TYPE "UDT_ModuleState"
TITLE = UDT_ModuleState
VERSION : 0.1
//User-defined structure of module states.
   STRUCT
      Configured { ExternalAccessible := 'False'; ExternalVisible := 'False'; ExternalWritable := 'False'} : Bool;   // Module configured
      Exist { ExternalAccessible := 'False'; ExternalVisible := 'False'; ExternalWritable := 'False'} : Bool;   // Module exist
      Error { ExternalAccessible := 'False'; ExternalVisible := 'False'; ExternalWritable := 'False'} : Bool;   // Module has error
   END_STRUCT;

END_TYPE

TYPE "UDT_DeviceState"
TITLE = UDT_DeviceState
VERSION : 0.1
//User-defined structure of device states.
   STRUCT
      Configure { ExternalAccessible := 'False'; ExternalVisible := 'False'; ExternalWritable := 'False'} : Bool;   // Device configured in TIA Portal hardware
      Exist { ExternalAccessible := 'False'; ExternalVisible := 'False'; ExternalWritable := 'False'} : Bool;   // Device physically connected
      Error { ExternalAccessible := 'False'; ExternalVisible := 'False'; ExternalWritable := 'False'} : Bool;   // Device has an error
      ProfinetNumber : UInt;   // Profinet slave number
      HW_ID : UInt;   // Device's HW_ID
      PNDeviceName : String;   // Device's project name
   END_STRUCT;

END_TYPE

TYPE "UDT_GINDHL"
VERSION : 0.1
   STRUCT
      ObjectID : String[10];   // Object ID
      VID : String[16];   // Virtual Item Identifier (VID)
      PieceID : String[40];   // Piece ID barcodes
      SortStrategy : String[1];   // Sort Strategy 1 - Highest priority available , 2 - Nearest
      ParcelReject { ExternalAccessible := 'False'; ExternalVisible := 'False'; ExternalWritable := 'False'} : Bool;   // True - Parcel reject
      Destination : Array[1..6] of Struct   // Destination
         ID : UInt;   // ID
         SortCommandActive { ExternalAccessible := 'False'; ExternalVisible := 'False'; ExternalWritable := 'False'} : Bool;   // Sort command
         ParcelSorted { ExternalAccessible := 'False'; ExternalVisible := 'False'; ExternalWritable := 'False'} : Bool;   // Parcel sorted
         Rejected { ExternalAccessible := 'False'; ExternalVisible := 'False'; ExternalWritable := 'False'} : Bool;   // Parcel rejected
         Reason : Int;   // Reason
      END_STRUCT;
      ParcelLocation : Struct   // Parcel Location
         Current : UInt;   // Current
         Last : UInt;   // Last
         Sort : UInt;   // Sort
      END_STRUCT;
      MFCMessage : Struct   // MFC Sort messages
         Sent : Struct   // Messages sent from the PLC to the MFC system
            SortResult { ExternalAccessible := 'False'; ExternalVisible := 'False'; ExternalWritable := 'False'} : Bool;   // Message Sort Result
            VIDResponse { ExternalAccessible := 'False'; ExternalVisible := 'False'; ExternalWritable := 'False'} : Bool;   // Message VID Response
            ScanReset { ExternalAccessible := 'False'; ExternalVisible := 'False'; ExternalWritable := 'False'} : Bool;   // Message Scan Reset
            XrayResult { ExternalAccessible := 'False'; ExternalVisible := 'False'; ExternalWritable := 'False'} : Bool;   // Message Xray result
            ParcelRegInfo { ExternalAccessible := 'False'; ExternalVisible := 'False'; ExternalWritable := 'False'} : Bool;   // Message Xray registration info
         END_STRUCT;
         Received : Struct   // Messages received from the MFC system to the PLC
            RejectParcel { ExternalAccessible := 'False'; ExternalVisible := 'False'; ExternalWritable := 'False'} : Bool;   // Message Reject Parcel
            Destination { ExternalAccessible := 'False'; ExternalVisible := 'False'; ExternalWritable := 'False'} : Bool;   // Message Destination
            DestinationResent { ExternalAccessible := 'False'; ExternalVisible := 'False'; ExternalWritable := 'False'} : Bool;   // Message Destination Resent
            TemporaryParcelIdentifier { ExternalAccessible := 'False'; ExternalVisible := 'False'; ExternalWritable := 'False'} : Bool;   // Message Temporary Parcel Identifier
            XrayRegistrationInfo { ExternalAccessible := 'False'; ExternalVisible := 'False'; ExternalWritable := 'False'} : Bool;
         END_STRUCT;
      END_STRUCT;
      Xray : Struct   // Xray data structure
         RoutingCode : String[2];   // Routing code
         Group : String[1];   // The group field is used to identify the group of the operator decisions came from in a
         Level : String[1];   // Level field is used to identify which level the operator decision came from in a
         Result : String[1];   // Results can be indicated with the following:A = Accept, R = Reject, U = Unavailable (Timeout), Z = High Threat
         BagIDMessage : Struct   // Message from PLC to Xray
            MessagePrepared { ExternalAccessible := 'False'; ExternalVisible := 'False'; ExternalWritable := 'False'} : Bool;   // The message is prepared and ready to send
            WrongMessageStructure { ExternalAccessible := 'False'; ExternalVisible := 'False'; ExternalWritable := 'False'} : Bool;   // The message has wrong structure
            Sent { ExternalAccessible := 'False'; ExternalVisible := 'False'; ExternalWritable := 'False'} : Bool;   // The message sent by PLC to Xray
            SentTime : String;   // Time when message sent by PLC to Xray
            NotSent { ExternalAccessible := 'False'; ExternalVisible := 'False'; ExternalWritable := 'False'} : Bool;   // The message was not sent from the PLC
            Received { ExternalAccessible := 'False'; ExternalVisible := 'False'; ExternalWritable := 'False'} : Bool;   // The message received by Xray
            TimeReceived : String;   // Time when message received by Xray
            NotReceived { ExternalAccessible := 'False'; ExternalVisible := 'False'; ExternalWritable := 'False'} : Bool;   // The message did not reach Xray
         END_STRUCT;
         DecisionMessage : Struct   // Message from Xray to PLC
            Received { ExternalAccessible := 'False'; ExternalVisible := 'False'; ExternalWritable := 'False'} : Bool;   // The message received by PLC
            ReceivedTime : String;   // The message received by PLC
            NotReceivedOnTime { ExternalAccessible := 'False'; ExternalVisible := 'False'; ExternalWritable := 'False'} : Bool;   // The message did not reach PLC
         END_STRUCT;
      END_STRUCT;
   END_STRUCT;

END_TYPE

TYPE "UDT_GINFedEx"
VERSION : 0.1
   STRUCT
      Timestamp : String[17];   // Local time timestamp
      TimeZoneDesignator : String[5];   // Time zone designator
      PackageEntrancePoint : String[14];   // Entrance point, where LLC starts tracking the parcel.
      PackageEntranceState : String[1];   // Entrance state
      PackageExitPoint : String[14];   // Exit point name, where LLC reports the last known tracking point.
      PackageExitState : String[1];   // Exit point state when LLC reports the last known tracking point.
      PalletType : String[2];   // Pallet code for different type of pallets on the market
      Mask : String[1];   // Flag to indicate that a pallet has been mask.
      CellNumber : String[4];   // Tray/Cell number (for loop sorters) or generated by LLC (on line sorters).
      CellsOccupied : String[1];   // Cells occupied by the piece for loop sorters.
      ImageID : String[6];   // Image ID number created by the ADC system.
      ScanUnitType : String[1];   // Scan unit type
      ADCSystemID : String[15];   // Number assigned by the ADC system
      PackageID : String[15];   // Number assigned by the LLC system
      LLCSystemID : String[15];
      HLCPackageID : String[10];   // Unique number for the specific package during it stays in HLC system.
      HLCResultCode : String[16];   // Result code based on processing of the scan event messages.
      ShipmentID : String[6];   // Consignment id of the parcel.
      WeightStatus : String[1];   // Status to indicate if the parcel/pallet has weight on the system.
      ActualDestination : String[6];   // Location code value that describes the actual disposition of the package.
      Destination1 : String[6];   // Location code value that describes where the package should go (Diverter Number).
      Destination2 : String[6];   // Location code value that describes where the package should go (Diverter Number).
      Destination3 : String[6];   // Location code value that describes where the package should go (Diverter Number).
      Destination4 : String[6];   // Location code value that describes where the package should go (Diverter Number).
      Destination5 : String[6];   // Location code value that describes where the package should go (Diverter Number).
      CutOffTimeDestination1 : String[5];   // Cut Off Time in Local Time.
      CutOffTimeDestination2 : String[5];   // Cut Off Time in Local Time.
      CutOffTimeDestination3 : String[5];   // Cut Off Time in Local Time.
      CutOffTimeDestination4 : String[5];   // Cut Off Time in Local Time.
      CutOffTimeDestination5 : String[5];   // Cut Off Time in Local Time.
      ReasonCode1 : String[8];   // Management Code value that describes the result of attempting to route the package to the Destination
      ReasonCode2 : String[8];   // Management Code value that describes the result of attempting to route the package to the Destination
      ReasonCode3 : String[8];   // Management Code value that describes the result of attempting to route the package to the Destination
      ReasonCode4 : String[8];   // Management Code value that describes the result of attempting to route the package to the Destination
      ReasonCode5 : String[8];   // Management Code value that describes the result of attempting to route the package to the Destination
      HLCDataText : String[20];   // Free text for future use.
      Customs : String[1];   // Need to be checked by customs
      DIMSystemID : String[15];   // Identifier of dimensioning system.
      DIMStatus : String[5];   // Basic diagnostic information from the dimensioning system at the moment of the measurement.
      PackageDimLength : String[6];   // Length dimension of package in resolution of dim system.
      PackageDimWidth : String[6];   // Width dimension of package in resolution of dim system.
      PackageDimHeight : String[6];   // Height dimension of package in resolution of dim system.
      DIMUOM : String[2];   // Unit of measure of the package dimensions.
      DimLFTstatusCode : String[8];   // Dimension LFT status code.
      DimConfidence : String[2];   // The level of assurance for the correct dimensions.
      DimensionSource : String[1];   // For combined camera/laser dim acquisition devices. It indicates type of capturing mode
      AlibiDims : String[25];   // Alibi for Dimensions
      SCLSystemID : String[15];   // Identifier of weight scale.
      SCLStatus : String[5];   // Basic diagnostic information from the weight scale system.
      SCLWT : String[6];   // Scale weight of package in resolution of scale system.
      SCLWTUOM : String[2];   // Unit of measurement for Weight
      SCLLFTStatusCode : String[2];   // Scale LFT status code.
      AlibiWeight : String[25];   // Alibi for Weight
      ReasonCode : String[1];   // This code should be used when the SI message has some defect.
      Stackable : String[1];   // If stackable recognition is enabled, Y or N
      Stickerstype : String[2];   // When optical recognition is used to sort
      FlyingDocument : String[1];   // Status to confirm if the document/flyer is prone to fly off the sorter.
      ModeofOperation : String[1];   // Camera Tunnel operational mode format:
      CameraHeadstatus : String[2];   // Diagnostic information on camera/laser heads performing barcode reads.
      PackageDataTruncated : String[1];   // Y = Full length of barcode data exceeds 9999 bytes, data truncated
      TotalBarcodeDataLength : String[4];   // Length of all barcode data that was sent in bytes;
      Barcode1Identification : String[3];   // Barcode identifier code.
      Barcode1status : String[2];   // Barcode confidence factor
      Barcode1datalength : String[4];   // String length of barcode data in bytes; inclusive of this field. Use 0054 as a fixed value
      Barcode1data : String[50];   // Highest priority barcode
      Barcode2Identification : String[3];   // Barcode identifier code.
      Barcode2status : String[2];   // Barcode confidence factor
      Barcode2datalength : String[4];   // String length of barcode data in bytes; inclusive of this field. Use 0054 as a fixed value
      Barcode2data : String[50];   // Highest priority barcode
      Barcode3Identification : String[3];   // Barcode identifier code.
      Barcode3status : String[2];   // Barcode confidence factor
      Barcode3datalength : String[4];   // String length of barcode data in bytes; inclusive of this field. Use 0054 as a fixed value
      Barcode3data : String[50];   // Highest priority barcode
      BarcodeIdentification : String[3];   // Barcode identifier code.
      Barcodestatus : String[2];   // Barcode confidence factor
      Barcodedatalength : String[4];   // String length of barcode data in bytes
      Barcodedata : String[50];   // Sortation barcode
      CustomerID : DInt;   // 6 digits SequentialID (NNNNNN)
      AreaNumber : String[2];   // Package Sequence ID "Area Number"
      PurgeEnabled { ExternalAccessible := 'False'; ExternalVisible := 'False'; ExternalWritable := 'False'} : Bool;   // Purge enabled for parcel: destination overwritten with Purge destination
   END_STRUCT;

END_TYPE

TYPE "UDT_GINStandard"
VERSION : 0.1
   STRUCT
      Destination : Array[0..20] of DInt;   // Destination
      Identification : Struct   // Barcode identification
         GoodRead { ExternalAccessible := 'False'; ExternalVisible := 'False'; ExternalWritable := 'False'} : Bool;   // Barcode read was succesful
         NoRead { ExternalAccessible := 'False'; ExternalVisible := 'False'; ExternalWritable := 'False'} : Bool;   // Barcode read was unsuccesful
         MultiRead { ExternalAccessible := 'False'; ExternalVisible := 'False'; ExternalWritable := 'False'} : Bool;   // Multiple Barcodes were detected
         Barcode : Array[0..10] of Char;   // Barcode values
      END_STRUCT;
      GinAssigned { ExternalAccessible := 'False'; ExternalVisible := 'False'; ExternalWritable := 'False'} : Bool;   // GIN is assigned to package
      Lost { ExternalAccessible := 'False'; ExternalVisible := 'False'; ExternalWritable := 'False'} : Bool;   // Lost in tracking
      Length : Int;   // Length in mm
      Width : Int;   // Width in mm
      Height : Int;   // Height in mm
      Weight : DInt;   // Weight in g
      PkgTooLong { ExternalAccessible := 'False'; ExternalVisible := 'False'; ExternalWritable := 'False'} : Bool;   // Package is too long
      PkgTooSmall { ExternalAccessible := 'False'; ExternalVisible := 'False'; ExternalWritable := 'False'} : Bool;   // Package is too small
      PkgTooHigh { ExternalAccessible := 'False'; ExternalVisible := 'False'; ExternalWritable := 'False'} : Bool;   // Package is too high
      PkgOverWeight { ExternalAccessible := 'False'; ExternalVisible := 'False'; ExternalWritable := 'False'} : Bool;   // Package is over weight
      TrailingGap : Int;   // Trailing gap size in cm between the package
      LeadingGap : Int;   // Leading gap size in cm between the package
      NrOfRecirculations : Int;   // Number of recirculations
      DestReqSend { ExternalAccessible := 'False'; ExternalVisible := 'False'; ExternalWritable := 'False'} : Bool;   // Destination request sent to high level
      DestRcv { ExternalAccessible := 'False'; ExternalVisible := 'False'; ExternalWritable := 'False'} : Bool;   // Destination received from high level
      SortStatus : Struct   // Sort status of the package
         DivertDestination : Int;   // Destination to which the package is diverted
         GoodDivert { ExternalAccessible := 'False'; ExternalVisible := 'False'; ExternalWritable := 'False'} : Bool;   // Package diverted
         FailedDivert { ExternalAccessible := 'False'; ExternalVisible := 'False'; ExternalWritable := 'False'} : Bool;   // Package failed to divert
         NoDivert : Bool := TRUE;   // Divert is not activated
         NoDivertCause : Struct   // Cause for no divert
            ChuteJam { ExternalAccessible := 'False'; ExternalVisible := 'False'; ExternalWritable := 'False'} : Bool;   // Chute is jammed
            ChuteFull { ExternalAccessible := 'False'; ExternalVisible := 'False'; ExternalWritable := 'False'} : Bool;   // Chute is full
            NoRTR { ExternalAccessible := 'False'; ExternalVisible := 'False'; ExternalWritable := 'False'} : Bool;   // Downstream conveyor is not ready to receive
            DestDisabled { ExternalAccessible := 'False'; ExternalVisible := 'False'; ExternalWritable := 'False'} : Bool;   // Destination is disabled
            TrayDisabled { ExternalAccessible := 'False'; ExternalVisible := 'False'; ExternalWritable := 'False'} : Bool;   // Tray is disabled
            SorterNotAtSpeed { ExternalAccessible := 'False'; ExternalVisible := 'False'; ExternalWritable := 'False'} : Bool;   // Sorter is not at speed
            LeadingGapError { ExternalAccessible := 'False'; ExternalVisible := 'False'; ExternalWritable := 'False'} : Bool;   // Gap size with downstream parcel is not enough
            TrailingGapError { ExternalAccessible := 'False'; ExternalVisible := 'False'; ExternalWritable := 'False'} : Bool;   // Gap size with upstream parcel is not enough
            PkgTooHigh { ExternalAccessible := 'False'; ExternalVisible := 'False'; ExternalWritable := 'False'} : Bool;   // Package is too high to divert
            PkgTooLong { ExternalAccessible := 'False'; ExternalVisible := 'False'; ExternalWritable := 'False'} : Bool;   // Package is too long to divert
            DestNotReachable { ExternalAccessible := 'False'; ExternalVisible := 'False'; ExternalWritable := 'False'} : Bool;   // Sort destionation is not reachable
            InvalidDest { ExternalAccessible := 'False'; ExternalVisible := 'False'; ExternalWritable := 'False'} : Bool;   // Sort destination is invalid
            DestTooLate { ExternalAccessible := 'False'; ExternalVisible := 'False'; ExternalWritable := 'False'} : Bool;   // Destination too late
            NoDestRcv { ExternalAccessible := 'False'; ExternalVisible := 'False'; ExternalWritable := 'False'} : Bool;   // Destination not received from high level
         END_STRUCT;
      END_STRUCT;
   END_STRUCT;

END_TYPE

TYPE "UDT_ProfinetDevice"
TITLE = UDT_ProfinetDevice
VERSION : 0.1
//User-defined structure of profinet device state.
   STRUCT
      DeviceState : "UDT_DeviceState";   // Device state
      Module { S7_SetPoint := 'False'} : Array[0..31] of "UDT_ModuleState";   // Modules
   END_STRUCT;

END_TYPE

TYPE "UDT_GINWCS"
VERSION : 0.1
   STRUCT
      ActionTaken : String;   // Location code value that describes the actual disposition of the package
      Destination1 : String[20];   // Location code value that describes where the package should go (Diverter Number)
      Destination2 : String[20];   // Location code value that describes where the package should go (Diverter Number)
      Destination3 : String[20];   // Location code value that describes where the package should go (Diverter Number)
      Destination4 : String[20];   // Location code value that describes where the package should go (Diverter Number)
      Destination5 : String[20];   // Location code value that describes where the package should go (Diverter Number)
      ReasonCode : String[2];   // Management Code value that describes the result of attempting to route the package to the Destination
      Barcode1 : String;   // Barcode identifier code
      Barcode2 : String;
      Barcode3 : String;
      Barcode4 : String;
   END_STRUCT;

END_TYPE

TYPE "UDT_GINWES"
VERSION : 0.1
   STRUCT
      Barcode : String[40];
   END_STRUCT;

END_TYPE

TYPE "UDT_GINUPS"
VERSION : 0.1
   STRUCT
      TRKNUM : String[18];   // Tracking number
      PKGUID : String[32];   // Package ID
      MSGID : String[32];   // Message ID
      Length : Int;   // Camera Length in mm
      Width : Int;   // Camera Width in mm
      Height : Int;   // Camera Height in mm
      Weight : DInt;   // Weight in g
      IDCreated { ExternalAccessible := 'False'; ExternalVisible := 'False'; ExternalWritable := 'False'} : Bool;   // Byte 1, Bit 0 - PLCID created or TrayID Read
      DimDataRcv { ExternalAccessible := 'False'; ExternalVisible := 'False'; ExternalWritable := 'False'} : Bool;   // Byte 1, Bit 1 - Package Dimensional Data Received via Camera Scan Data Message
      PkgWrongInduct { ExternalAccessible := 'False'; ExternalVisible := 'False'; ExternalWritable := 'False'} : Bool;   // Byte 1, Bit 2 - Package Did NOT Induct Properly (Non-Tray Systems)
      IDCalcFromCamID { ExternalAccessible := 'False'; ExternalVisible := 'False'; ExternalWritable := 'False'} : Bool;   // Byte 2, Bit 0 - PLCID/TrayID Calculated From CamID
      UnknownParcelID { ExternalAccessible := 'False'; ExternalVisible := 'False'; ExternalWritable := 'False'} : Bool;   // Byte 2, Bit 4 - Unknown Parcel ID
      UndefinedProblem { ExternalAccessible := 'False'; ExternalVisible := 'False'; ExternalWritable := 'False'} : Bool;   // Byte 2, Bit 5 - Un-Defined Problem
      UnrecognizedCmd { ExternalAccessible := 'False'; ExternalVisible := 'False'; ExternalWritable := 'False'} : Bool;   // Byte 2, Bit 6 - Un-recognized command
      SorterInMainteneceMode { ExternalAccessible := 'False'; ExternalVisible := 'False'; ExternalWritable := 'False'} : Bool;   // Byte 2, Bit 7 - Sorter in Maintenance/Commissioning Mode
      DestUserSusp { ExternalAccessible := 'False'; ExternalVisible := 'False'; ExternalWritable := 'False'} : Bool;   // Byte 3, Bit 3 - Destination User Suspended
      SorterNotSynch { ExternalAccessible := 'False'; ExternalVisible := 'False'; ExternalWritable := 'False'} : Bool;   // Byte 3, Bit 6 - Sorter NOT Synchronized (Tilt Tray Systems)
      PkgDetAtVerCheckPoint { ExternalAccessible := 'False'; ExternalVisible := 'False'; ExternalWritable := 'False'} : Bool;   // Byte 4, Bit 0 - Package Detected at Verification Check Point
      ChuteFullAftrAlterDest { ExternalAccessible := 'False'; ExternalVisible := 'False'; ExternalWritable := 'False'} : Bool;   // Byte 4, Bit 7 - Preferred chute full after passed alternate destination
      ChuteNotAvailAfterAlterDest { ExternalAccessible := 'False'; ExternalVisible := 'False'; ExternalWritable := 'False'} : Bool;   // Byte 5, Bit 0 - Preferred chute not available after passed alternate destination
      PLCRedirected { ExternalAccessible := 'False'; ExternalVisible := 'False'; ExternalWritable := 'False'} : Bool;   // Byte 5, Bit 2 - PLC Redirected
      ThreatParcel { ExternalAccessible := 'False'; ExternalVisible := 'False'; ExternalWritable := 'False'} : Bool;   // Threat parcel
   END_STRUCT;

END_TYPE

DATA_BLOCK "DB_Memory"
TITLE = DB_Memory
{ S7_Optimized_Access := 'TRUE' }
AUTHOR : MHSE
VERSION : 3.0
NON_RETAIN
   VAR
      ClockByte { ExternalAccessible := 'False'; ExternalVisible := 'False'; ExternalWritable := 'False'} : Byte;   // System clock byte
      Clock_10Hz { ExternalAccessible := 'False'; ExternalVisible := 'False'; ExternalWritable := 'False'} : Bool;   // 10 Hz system clock bit
      Clock_5Hz { ExternalAccessible := 'False'; ExternalVisible := 'False'; ExternalWritable := 'False'} : Bool;   // 5 Hz system clock bit
      "Clock_2.5Hz" { ExternalAccessible := 'False'; ExternalVisible := 'False'; ExternalWritable := 'False'} : Bool;   // 2.5 Hz system clock bit
      Clock_2Hz { ExternalAccessible := 'False'; ExternalVisible := 'False'; ExternalWritable := 'False'} : Bool;   // 2 Hz system clock bit
      "Clock_1.25Hz" { ExternalAccessible := 'False'; ExternalVisible := 'False'; ExternalWritable := 'False'} : Bool;   // 1.25 Hz system clock bit
      Clock_1Hz { ExternalAccessible := 'False'; ExternalVisible := 'False'; ExternalWritable := 'False'} : Bool;   // 1 Hz system clock bit
      "Clock_0.625Hz" { ExternalAccessible := 'False'; ExternalVisible := 'False'; ExternalWritable := 'False'} : Bool;   // 0.625 Hz system clock bit
      "Clock_0.5Hz" { ExternalAccessible := 'False'; ExternalVisible := 'False'; ExternalWritable := 'False'} : Bool;   // 0.5 Hz system clock bit
      SystemByte { ExternalAccessible := 'False'; ExternalVisible := 'False'; ExternalWritable := 'False'} : Byte;   // System byte
      OSClockByte { ExternalAccessible := 'False'; ExternalVisible := 'False'; ExternalWritable := 'False'} : Byte;   // One shot of clock pulse
      "OS_0.1sec" { ExternalAccessible := 'False'; ExternalVisible := 'False'; ExternalWritable := 'False'} : Bool;   // One shot every 0.1 sec
      "OS_0.2sec" { ExternalAccessible := 'False'; ExternalVisible := 'False'; ExternalWritable := 'False'} : Bool;   // One shot every 0.2 sec
      "OS_0.4sec" { ExternalAccessible := 'False'; ExternalVisible := 'False'; ExternalWritable := 'False'} : Bool;   // One shot every 0.4 sec
      "OS_0.5sec" { ExternalAccessible := 'False'; ExternalVisible := 'False'; ExternalWritable := 'False'} : Bool;   // One shot every 0.5 sec
      "OS_0.8sec" { ExternalAccessible := 'False'; ExternalVisible := 'False'; ExternalWritable := 'False'} : Bool;   // One shot every 0.8 sec
      OS_1sec { ExternalAccessible := 'False'; ExternalVisible := 'False'; ExternalWritable := 'False'} : Bool;   // One shot every 1 sec
      "OS_1.6sec" { ExternalAccessible := 'False'; ExternalVisible := 'False'; ExternalWritable := 'False'} : Bool;   // One shot every 1.6 sec
      OS_2sec { ExternalAccessible := 'False'; ExternalVisible := 'False'; ExternalWritable := 'False'} : Bool;   // One shot every 2 sec
      PrevCycleTime { ExternalAccessible := 'False'; ExternalVisible := 'False'; ExternalWritable := 'False'} : LReal;   // Previous PLC cycle Time
      RuntimeMem { ExternalAccessible := 'False'; ExternalVisible := 'False'; ExternalWritable := 'False'} : LReal;   // Runtime memory
      FirstScan { ExternalAccessible := 'False'; ExternalVisible := 'False'; ExternalWritable := 'False'} : Bool;   // First scan bit
      DiagStatusUpdate { ExternalAccessible := 'False'; ExternalVisible := 'False'; ExternalWritable := 'False'} : Bool;   // Diagnostic status update
      AlwaysTrue { ExternalAccessible := 'False'; ExternalVisible := 'False'; ExternalWritable := 'False'} : Bool;   // Always True bit
      AlwaysFalse { ExternalAccessible := 'False'; ExternalVisible := 'False'; ExternalWritable := 'False'} : Bool;   // Always False bit
      CommissioningFalse { ExternalAccessible := 'False'; ExternalVisible := 'False'; ExternalWritable := 'False'} : Bool;   // Commissioning always false
      CommissioningTrue { ExternalAccessible := 'False'; ExternalVisible := 'False'; ExternalWritable := 'False'} : Bool;   // Commissioning always true
      ReconnectCommand { ExternalAccessible := 'False'; ExternalVisible := 'False'; ExternalWritable := 'False'} : Bool;   // Reconnect command
      ScanMainRack { ExternalAccessible := 'False'; ExternalVisible := 'False'; ExternalWritable := 'False'} : Bool;   // Trigger to check main rack confiuration
      ScanProfinet { ExternalAccessible := 'False'; ExternalVisible := 'False'; ExternalWritable := 'False'} : Bool;   // Scan profinet bit
      Simulation { ExternalAccessible := 'False'; ExternalVisible := 'False'; ExternalWritable := 'False'} : Bool;   // Simulation
      PN1OK { ExternalAccessible := 'False'; ExternalVisible := 'False'; ExternalWritable := 'False'} : Bool;   // Profinet ok
      "Local~PROFINET_IO-System" { ExternalAccessible := 'False'; ExternalVisible := 'False'; ExternalWritable := 'False'} : HW_ANY;   // HW Intentifier of PN-IO System
      "Local~PROFINET_IO-System_1" { ExternalAccessible := 'False'; ExternalVisible := 'False'; ExternalWritable := 'False'} : HW_ANY;   // HW Intentifier of PN-IOSystem 1
      "Local~PROFINET_IO-System_2" { ExternalAccessible := 'False'; ExternalVisible := 'False'; ExternalWritable := 'False'} : HW_ANY;   // HW Intentifier of PN-IOSystem 2
      "Local~PROFINET_IO-System_3" { ExternalAccessible := 'False'; ExternalVisible := 'False'; ExternalWritable := 'False'} : HW_ANY;   // HW Intentifier of PN-IOSystem 3
      "Local~PROFINET_IO-System_4" { ExternalAccessible := 'False'; ExternalVisible := 'False'; ExternalWritable := 'False'} : HW_ANY;   // HW Intentifier of PN-IOSystem 4
      "Local~PROFINET_IO-System_5" { ExternalAccessible := 'False'; ExternalVisible := 'False'; ExternalWritable := 'False'} : HW_ANY;   // HW Intentifier of PN-IOSystem 5
      "Local~PROFINET_IO-System_6" { ExternalAccessible := 'False'; ExternalVisible := 'False'; ExternalWritable := 'False'} : HW_ANY;   // HW Intentifier of PN-IOSystem 6
      "Local~PROFINET_IO-System_7" { ExternalAccessible := 'False'; ExternalVisible := 'False'; ExternalWritable := 'False'} : HW_ANY;   // HW Intentifier of PN-IOSystem 7
      "Local~PROFINET_IO-System_8" { ExternalAccessible := 'False'; ExternalVisible := 'False'; ExternalWritable := 'False'} : HW_ANY;   // HW Intentifier of PN-IOSystem 8
      "Local~PROFINET_IO-System_9" { ExternalAccessible := 'False'; ExternalVisible := 'False'; ExternalWritable := 'False'} : HW_ANY;   // HW Intentifier of PN-IOSystem 9
   END_VAR


BEGIN

END_DATA_BLOCK

TYPE "UDT_GIN"
VERSION : 0.1
   STRUCT
      General { S7_SetPoint := 'False'} : "UDT_GINStandard";
      FedEx { S7_SetPoint := 'False'} : "UDT_GINFedEx";
      UPS { S7_SetPoint := 'False'} : "UDT_GINUPS";
      DHL { S7_SetPoint := 'False'} : "UDT_GINDHL";
      WCS { S7_SetPoint := 'False'} : "UDT_GINWCS";
      WES { S7_SetPoint := 'False'} : "UDT_GINWES";
   END_STRUCT;

END_TYPE

TYPE "UDT_FifoStatus"
TITLE = UDT_FifoStatus
VERSION : 0.1
//
//User-defined structure of FC_Fifo function status.
//Version History:
//Date              | Version   | Author         | Remark
//24/05/2019  | 0.1           | K.Pokorski   | first release MHSE TIA 15.1
//24/05/2019  | 0.2           | K.Pokorski   | first release MHSE TIA 15.1
//
   STRUCT
      InvalidMode { ExternalAccessible := 'False'; ExternalVisible := 'False'; ExternalWritable := 'False'} : Bool;   // Invalid mode selected
      InvalidMaxNrOfEntries { ExternalAccessible := 'False'; ExternalVisible := 'False'; ExternalWritable := 'False'} : Bool;   // Invalid maximum number of entries or buffer is not an array
      InvalidTotalEntriesStored { ExternalAccessible := 'False'; ExternalVisible := 'False'; ExternalWritable := 'False'} : Bool;   // Invalid total number of entries
      InvalidNextEntryToWrite { ExternalAccessible := 'False'; ExternalVisible := 'False'; ExternalWritable := 'False'} : Bool;   // Invalid number of next entry to write
      InvalidNextEntryToRead { ExternalAccessible := 'False'; ExternalVisible := 'False'; ExternalWritable := 'False'} : Bool;   // Invalid number of next entry to read
      InvalidDataType { ExternalAccessible := 'False'; ExternalVisible := 'False'; ExternalWritable := 'False'} : Bool;   // Message and buffer element data type inconsistent
      FifoPreFull { ExternalAccessible := 'False'; ExternalVisible := 'False'; ExternalWritable := 'False'} : Bool;   // 90 % of FIFO data buffer capacity reached
      FifoFull { ExternalAccessible := 'False'; ExternalVisible := 'False'; ExternalWritable := 'False'} : Bool;   // FIFO data buffer full
   END_STRUCT;

END_TYPE

TYPE "UDT_ProfinetNetwork"
TITLE = UDT_ProfinetNetwork
VERSION : 0.1
//User-defined structure of profinet network state.
   STRUCT
      DeviceStatus : Array[0..512] of "UDT_ProfinetDevice";   // Profinet device status
   END_STRUCT;

END_TYPE

TYPE "UDT_FifoHeader"
TITLE = UDT_FifoHeader
VERSION : 0.1
//User-defined structure of FIFO register header information.
   STRUCT
      Status : Struct   // Status bits
         Empty { ExternalAccessible := 'False'; ExternalVisible := 'False'; ExternalWritable := 'False'} : Bool;   // FIFO Empty
         Prefull { ExternalAccessible := 'False'; ExternalVisible := 'False'; ExternalWritable := 'False'} : Bool;   // FIFO Prefull
         Full { ExternalAccessible := 'False'; ExternalVisible := 'False'; ExternalWritable := 'False'} : Bool;   // FIFO Full
      END_STRUCT;
      NextEntryToRead : Int;   // Next FIFO entry to read
      NextEntryToWrite : Int;   // Next FIFO entry to write
      MaxNrOfEntries : Int;   // Maximum number of FIFO entries
      TotalEntriesStored : Int;   // Total number of FIFO entries
   END_STRUCT;

END_TYPE

FUNCTION "FC_GetNrOfArrayEl" : Int
TITLE = FC_GetNrOfArrayEl
{ S7_Optimized_Access := 'TRUE' }
AUTHOR : MHSE
FAMILY : GeneralSystemFunctions
VERSION : 3.0
// ATTRIBUTES
// AUTO_NUMBER = True
// BLOCK_NUMBER = 19
// END_ATTRIBUTES
//Function to get the number of array elements.
   VAR_INPUT
      iv_Array : Variant;   // Input array
   END_VAR

   VAR_TEMP
      ti_NrOfArrayEl : Int;   // Number of array elements
   END_VAR


BEGIN
	(*
	----------------------------------------------------------------------------------------

	Version history:
	Date        | Version   | Author        | Remark
	----------------------------------------------------------------------------------------
	24/05/2019  | 0.1       | L.Klar        | first release MHS TIA 15.1
	24/07/2019  | 2.0       | L.Klar        | 2.0 MHS library release TIA 15.1
	27/08/2019  | 2.1       | K.Pokorski    | Comments adjusted
	12/11/2019  | 3.0       | P.Majka       | 3.0 MHS library release TIA 15.1
	21/02/2023  | 4.0       | F.Baten       | 4.0 Release TIA 17.5
	*)

	REGION 1 – Number of an array elements

	    IF IS_ARRAY(#iv_Array)                                                  // Input variable is an array
	    THEN

	        #ti_NrOfArrayEl := UDINT_TO_INT(CountOfElements(#iv_Array));

	        // Reset array length if the input variable isn't an array
	    ELSE

	        #ti_NrOfArrayEl := 0;

	    END_IF;

	END_REGION

	REGION 2 – Return output

	    #FC_GetNrOfArrayEl := #ti_NrOfArrayEl;

	END_REGION

END_FUNCTION

TYPE "UDT_CommonStatus"
TITLE = UDT_CommonStatus
VERSION : 0.1
//User-defined structure of common statuses.
   STRUCT
      SafetyStop { ExternalAccessible := 'False'; ExternalVisible := 'False'; ExternalWritable := 'False'} : Bool;   // Emergancy stop
      Error { ExternalAccessible := 'False'; ExternalVisible := 'False'; ExternalWritable := 'False'} : Bool;   // An error is active
      Warning { ExternalAccessible := 'False'; ExternalVisible := 'False'; ExternalWritable := 'False'} : Bool;   // A warning is active
      ManualRun { ExternalAccessible := 'False'; ExternalVisible := 'False'; ExternalWritable := 'False'} : Bool;   // Running in manual mode
      Manual { ExternalAccessible := 'False'; ExternalVisible := 'False'; ExternalWritable := 'False'} : Bool;   // In manual mode
      Halted { ExternalAccessible := 'False'; ExternalVisible := 'False'; ExternalWritable := 'False'} : Bool;   // Halted
      Dieback { ExternalAccessible := 'False'; ExternalVisible := 'False'; ExternalWritable := 'False'} : Bool;   // In dieback
      Stopped { ExternalAccessible := 'False'; ExternalVisible := 'False'; ExternalWritable := 'False'} : Bool;   // Stopped
      Running { ExternalAccessible := 'False'; ExternalVisible := 'False'; ExternalWritable := 'False'} : Bool;   // Running
      EnergySave { ExternalAccessible := 'False'; ExternalVisible := 'False'; ExternalWritable := 'False'} : Bool;   // In energy saving mode
      AutoON { ExternalAccessible := 'False'; ExternalVisible := 'False'; ExternalWritable := 'False'} : Bool;   // Automatic started
   END_STRUCT;

END_TYPE

TYPE "UDT_EventStatistic"
TITLE = UDT_EventStatistic
VERSION : 0.1
//User-defined structure of event statistic data.
   STRUCT
      NumberOfTimes : DInt;   // Number of times the event occurred since last reset
      LastEventSeconds : DInt;   // Number of seconds of the current or last event
      TotalEventSeconds : DInt;   // Total number of seconds the event occurred since last reset
   END_STRUCT;

END_TYPE

DATA_BLOCK "DB_Time"
TITLE = DB_Time
{ S7_Optimized_Access := 'TRUE' }
AUTHOR : MHSE
FAMILY : GeneralSystemFunctions
VERSION : 3.0
NON_RETAIN
//Data block to store date and time data.
   VAR
      ActualTimeDTL {InstructionName := 'DTL'; LibVersion := '1.0'; ExternalAccessible := 'False'; ExternalVisible := 'False'; ExternalWritable := 'False'} : DTL;   // Actual date and time in DTL
      ActualTime { ExternalAccessible := 'False'; ExternalVisible := 'False'; ExternalWritable := 'False'} : String;   // Actual date and time in String
      Timestamp { ExternalAccessible := 'False'; ExternalVisible := 'False'; ExternalWritable := 'False'} : String[17];   // Actual date and time in String
      DaylightSaving { ExternalAccessible := 'False'; ExternalVisible := 'False'; ExternalWritable := 'False'} : Int;
   END_VAR


BEGIN

END_DATA_BLOCK

TYPE "UDT_EquipmentControl"
TITLE = UDT_EquipmentControl
VERSION : 0.1
//User-defined structure of equipment control commands.
   STRUCT
      Command : Struct   // Control command
         Start { ExternalAccessible := 'False'; ExternalVisible := 'False'; ExternalWritable := 'False'} : Bool;   // Start conveyor
         Stop { ExternalAccessible := 'False'; ExternalVisible := 'False'; ExternalWritable := 'False'} : Bool;   // Stop conveyor
         Reset { ExternalAccessible := 'False'; ExternalVisible := 'False'; ExternalWritable := 'False'} : Bool;   // Faults reset
         ResetData { ExternalAccessible := 'False'; ExternalVisible := 'False'; ExternalWritable := 'False'} : Bool;   // Statistics reset
         ManualMode { ExternalAccessible := 'False'; ExternalVisible := 'False'; ExternalWritable := 'False'} : Bool;   // Manual mode required
         DisableManualMode { ExternalAccessible := 'False'; ExternalVisible := 'False'; ExternalWritable := 'False'} : Bool;   // Disable manual mode
         AutomaticOn { ExternalAccessible := 'False'; ExternalVisible := 'False'; ExternalWritable := 'False'} : Bool;   // System is started in automatic mode
         StopRequest { ExternalAccessible := 'False'; ExternalVisible := 'False'; ExternalWritable := 'False'} : Bool;
      END_STRUCT;
      Report { S7_SetPoint := 'False'} : "UDT_CommonStatus";   // Conveyors state
      Request : Struct   // Request from equipment
         RestartRequired { ExternalAccessible := 'False'; ExternalVisible := 'False'; ExternalWritable := 'False'} : Bool;   // Restart required from system control
         SignalingRequest { ExternalAccessible := 'False'; ExternalVisible := 'False'; ExternalWritable := 'False'} : Bool;   // Beeper required
         InhibitStop { ExternalAccessible := 'False'; ExternalVisible := 'False'; ExternalWritable := 'False'} : Bool;
      END_STRUCT;
   END_STRUCT;

END_TYPE

TYPE "UDT_VfdKebaSystemSpeedAxisConfiguration"
VERSION : 0.1
   STRUCT
      BeltSpeedCorrection : Int := 100;   // Belt speed correction [%]
      Acceleration : UInt;   // VFD ramp up time for monitoring starting [mm/s2]
      Deceleration : UInt;   // VFD ramp up time for monitoring stopping [mm/s2]
      SpeedSetpointWindow : Int := 5;   // VFD speed setpoint window (tolerance) [mm/s]
      DirectionReversal : Bool;   // If true, direction will be swapped
      InterlockFwd : Bool := TRUE;   // False when turning in forward direction is not possible / allowed
      InterlockRvs : Bool := TRUE;   // False when turning in reverse direction is not possible / allowed
   END_STRUCT;

END_TYPE

TYPE "UDT_PNDevice"
VERSION : 0.1
   STRUCT
      PNNetworknumber : Int := 1;   // Number of the profinet network where device exist
      PNDeviceNumber : Int := 0;   // Profinet number of the device
      PNDeviceFound { ExternalAccessible := 'False'; ExternalVisible := 'False'; ExternalWritable := 'False'} : Bool;   // Device found in Profinet structure
   END_STRUCT;

END_TYPE

DATA_BLOCK "DB_ProfinetDiagnostic"
TITLE = DB_ProfinetDiagnostic
{ S7_Optimized_Access := 'TRUE' }
AUTHOR : MHSE
FAMILY : GeneralSystemFunctions
VERSION : 3.0
NON_RETAIN
//Data block to store profinet network diagnostic data.
   VAR
      ProfinetNetworks { ExternalAccessible := 'False'; ExternalVisible := 'False'; ExternalWritable := 'False'; S7_SetPoint := 'False'} : Array[1..10] of "UDT_ProfinetNetwork";
   END_VAR


BEGIN

END_DATA_BLOCK

FUNCTION_BLOCK "FB_TimerOnOffDelay"
TITLE = FB_TimerOnOffDelay
{ S7_Optimized_Access := 'TRUE' }
AUTHOR : MHSE
FAMILY : GeneralSystemFunctions
VERSION : 3.0
// ATTRIBUTES
// AUTO_NUMBER = True
// BLOCK_NUMBER = 32
// END_ATTRIBUTES
//Function block to generate on/off signal delay.
   VAR_INPUT
      iudi_OnDelayTime { ExternalAccessible := 'False'; ExternalVisible := 'False'; ExternalWritable := 'False'} : UDInt;   // On delay time [ms]
      iudi_OffDelayTime { ExternalAccessible := 'False'; ExternalVisible := 'False'; ExternalWritable := 'False'} : UDInt;   // Off delay time [ms]
      ix_SignalToDelay { ExternalAccessible := 'False'; ExternalVisible := 'False'; ExternalWritable := 'False'} : Bool;   // Input signal to be delayed
      ix_Enable { ExternalAccessible := 'False'; ExternalVisible := 'False'; ExternalWritable := 'False'} : Bool := TRUE;   // Timer Enable
   END_VAR

   VAR_OUTPUT
      qlr_ActualTime { ExternalAccessible := 'False'; ExternalVisible := 'False'; ExternalWritable := 'False'} : LReal;   // Actual time
      qx_DelayedSignal { ExternalAccessible := 'False'; ExternalVisible := 'False'; ExternalWritable := 'False'} : Bool;   // Delayed signal output
   END_VAR

   VAR
      s_R_TRIG_Signal {InstructionName := 'R_TRIG'; LibVersion := '1.0'; ExternalAccessible := 'False'; ExternalVisible := 'False'; ExternalWritable := 'False'; S7_SetPoint := 'False'} : R_TRIG;   // Siemens "R_Trig" - to prepare the rising edge trigger on "ix_SignalToDelay" signal
      s_F_TRIG_Signal {InstructionName := 'F_TRIG'; LibVersion := '1.0'; ExternalAccessible := 'False'; ExternalVisible := 'False'; ExternalWritable := 'False'; S7_SetPoint := 'False'} : F_TRIG;   // Siemens "F_Trig" - to prepare the falling edge trigger on "ix_SignalToDelay" signal
   END_VAR
   VAR RETAIN
      slr_ActualDelayTime { ExternalAccessible := 'False'; ExternalVisible := 'False'; ExternalWritable := 'False'} : LReal;   // Actual delay time [ms]
   END_VAR


BEGIN
	(*
	----------------------------------------------------------------------------------------

	Version history:
	Date        | Version   | Author        | Remark
	----------------------------------------------------------------------------------------
	24/05/2019  | 0.1       | L.Klar        | first release MHS TIA 15.1
	24/07/2019  | 2.0       | L.Klar        | 2.0 MHS library release TIA 15.1
	26/08/2019  | 2.1       | M.Kurpiers    | Comments adjusted
	04/11/2019  | 2.2       | L.Klar        | Prevoius cycle scan changed from memory to DB variable
	12/11/2019  | 3.0       | P.Majka       | 3.0 MHS library release TIA 15.1
	21/02/2023  | 4.0       | F.Baten       | 4.0 Release TIA 17.5
	*)

	REGION Step 1 – Input signal edge detection

	    #s_R_TRIG_Signal(CLK := #ix_SignalToDelay);


	    #s_F_TRIG_Signal(CLK := #ix_SignalToDelay);

	END_REGION

	REGION Step 2 – Actual delay time initialization

	    IF (#s_R_TRIG_Signal.Q OR #s_F_TRIG_Signal.Q)           // Input signal changed
	    THEN

	        #slr_ActualDelayTime := 0;

	    END_IF;

	END_REGION

	REGION Step 3 – On/Off delay time calculation


	    IF (#ix_SignalToDelay                                       // Signal to be delayed is active
	        AND #ix_Enable)                                         // Ttimer enabled
	    THEN

	        // Timer on
	        IF (#slr_ActualDelayTime >= #iudi_OnDelayTime)
	        THEN

	            #qx_DelayedSignal := TRUE;

	        ELSE

	            #slr_ActualDelayTime += "DB_Memory".PrevCycleTime;

	        END_IF;

	    END_IF;

	    // Timer off
	    IF (NOT #ix_SignalToDelay                                   // Signal to delay is not active
	        AND #ix_Enable)                                         // Timer is enabled
	    THEN

	        IF (#slr_ActualDelayTime >= #iudi_OffDelayTime)
	        THEN

	            #qx_DelayedSignal := FALSE;

	        ELSE

	            #slr_ActualDelayTime += "DB_Memory".PrevCycleTime;

	        END_IF;

	    END_IF;

	END_REGION

	REGION Step 4 – Actual time

	    #qlr_ActualTime := #slr_ActualDelayTime;

	END_REGION
END_FUNCTION_BLOCK

TYPE "UDT_FedExFacility"
VERSION : 0.1
   STRUCT
      FacilityID : String := '';   // Generated during configuration. It is a fixed value for all systems.
      SystemID : String;   // System ID of the system making the request.
      System : Struct   // System information
         LOC : String;
         TYP : String;
         Number : String;
      END_STRUCT;
      VersionID : String;   // Interface document version.
      TimeZoneDesignator : String;   // Time Zone Designator
      SS : UDInt;   // Maximum frequency of the messages
   END_STRUCT;

END_TYPE

TYPE "UDT_VfdKebaSystemPositioningAxisConfiguration"
VERSION : 0.1
   STRUCT
      PositionWindow : Int;   // Position window (tolerance) [degree]
      PositionMax : Int;   // Maximum allowed position [degree]
      PositionMin : Int;   // Minimum allowed position [degree]
      VFDSpeed : Int;   // Speed to run in automatic mode [degree/s]
      Position : Array[0..10] of Int;   // Positions in degree's to move to as requested
   END_STRUCT;

END_TYPE

TYPE "UDT_StopRollerConfiguration"
VERSION : 0.1
   STRUCT
      BrakePuls : UDInt;   // Time [ms] brake is up in brake function
      BrakePause : UDInt;   // Time [ms] brake is down in brake function
      BrakePauseLong : UDInt;   // Long time [ms] brake is down in brake function
      PECBrakeOnDelay : UDInt;   // On delay time PEC brake signal
      PECBrakeOffDelay : UDInt;   // Off delay time PEC brake signal
      PECStopOnDelay : UDInt;   // On delay time PEC stop signal
      PECStopOffDelay : UDInt;   // Off delay time PEC stop signal
      StopFunctionOnDelay : UDInt;   // On delay time stop function
      StopFunctionOffDelay : UDInt;   // Off delay time stop function
      FailSafe { ExternalAccessible := 'False'; ExternalVisible := 'False'; ExternalWritable := 'False'} : Bool;   // Activate output to release
   END_STRUCT;

END_TYPE

TYPE "UDT_PneumaticBrakeConfiguration"
VERSION : 0.1
   STRUCT
      BrakePuls : UDInt;   // Time [ms] brake is up in brake function
      BrakePause : UDInt;   // Time [ms] brake is down in brake function
      BrakeCycles : Int;   // Number of brake cycles
      BrakeInterval : UDInt;   // Time [ms] between brake cycles
      PECBrakeOnDelay : UDInt;   // On delay time PEC brake signal
      PECBrakeOffDelay : UDInt;   // Off delay time PEC brake signal
      PECStopOnDelay : UDInt;   // On delay time PEC stop signal
      PECStopOffDelay : UDInt;   // Off delay time PEC stop signal
      StopFunctionOnDelay : UDInt;   // On delay time stop function
      StopFunctionOffDelay : UDInt;   // Off delay time stop function
      FailSafe { ExternalAccessible := 'False'; ExternalVisible := 'False'; ExternalWritable := 'False'} : Bool;   // Activate output to release
      Slave { ExternalAccessible := 'False'; ExternalVisible := 'False'; ExternalWritable := 'False'} : Bool;   // Stopper is slave
   END_STRUCT;

END_TYPE

FUNCTION "FC_Fifo" : Void
TITLE = FC_Fifo
{ S7_Optimized_Access := 'TRUE' }
AUTHOR : MHSE
FAMILY : GeneralSystemFunctions
VERSION : 3.0
// ATTRIBUTES
// AUTO_NUMBER = True
// BLOCK_NUMBER = 17
// END_ATTRIBUTES
//Function for controlling FIFO register.
   VAR_INPUT
      ic_Mode : Char;   // Mode selector: "W" - Write; "R" - Read; "C" - Clear (Reset) "S" - Status
   END_VAR

   VAR_OUTPUT
      qUDT_Status : "UDT_FifoStatus";   // FIFO status structure
      qx_Error : Bool;   // Collective error output
      qx_Warning : Bool;   // Collective warning output
   END_VAR

   VAR_IN_OUT
      iqv_Data : Variant;   // Data
      iqUDT_FifoHeader : "UDT_FifoHeader";   // FIFO header
      iqv_DataBuffer : Variant;   // FIFO data buffer
   END_VAR

   VAR_TEMP
      tUDT_Status : "UDT_FifoStatus";   // Status structure
      ti_MoveBLKErrorCode : Int;   // Move_BLK_Variant function return
      tx_HeaderValid : Bool;   // Header valid
   END_VAR


BEGIN
	(*
	----------------------------------------------------------------------------------------

	Version history:
	Date        | Version   | Author        | Remark
	----------------------------------------------------------------------------------------
	24/05/2019  | 0.1       | L.Klar        | first release MHS TIA 15.1
	14/06/2019  | 0.2       | A.Nowak       | Replacement of instruction if for direct write into variable - Region 3 , 4.1 , 4.2 , 4.3 , 4.4 , 8.1  , 8.2
	17/07/2019  | 0.3       | L.Klar        | Status handling changed
	24/07/2019  | 2.0       | L.Klar        | 2.0 MHS library release TIA 15.1
	23/08/2019  | 2.1       | K.Pokorski    | Comments corrected
	27/08/2019  | 2.2       | M.Kurpiers    | Comments adjusted
	27/09/2019  | 2.3       | K.Pokorski    | Variant input included
	01/10/2019  | 2.4       | A.Nowak       | Correct comments and rename regions
	12/11/2019  | 3.0       | P.Majka       | 3.0 MHS library release TIA 15.1
	21/02/2023  | 4.0       | F.Baten       | 4.0 Release TIA 17.5
	*)

	REGION 1 – Diagnostic bits initialization

	    // Clear FIFO statuses
	    #tUDT_Status.FifoFull := FALSE;
	    #tUDT_Status.FifoPreFull := FALSE;

	END_REGION

	REGION 2 – Array's information

	    // If buffer elements type is invalid, set the error
	    #tUDT_Status.InvalidDataType := NOT (TypeOf(#iqv_Data) = TypeOfElements(#iqv_DataBuffer));

	END_REGION

	REGION 3 – Mode validation

	    // Set the mode invalid if selected mode isn't one of the following: W- Write, R - Read, C - Clear, S - Status
	    #tUDT_Status.InvalidMode := #ic_Mode <> 'W'
	    AND #ic_Mode <> 'R'
	    AND #ic_Mode <> 'C'
	    AND #ic_Mode <> 'S';

	END_REGION

	REGION 4 – The header settings checking

	    // The correct mode has been selected and data type is valid
	    IF (NOT #tUDT_Status.InvalidMode
	        AND NOT #tUDT_Status.InvalidDataType)
	    THEN

	        REGION 4.1 – The number of maximum FIFO entries validation

	            // Write the number of array's elements to FIFO header
	            #iqUDT_FifoHeader.MaxNrOfEntries := "FC_GetNrOfArrayEl"(#iqv_DataBuffer);

	            // Set the invalid maximum number of entries error
	            #tUDT_Status.InvalidMaxNrOfEntries := #iqUDT_FifoHeader.MaxNrOfEntries <= 0;

	        END_REGION

	        REGION 4.2 – The number of total FIFO entries validation

	            // Set the invalid total number of entries error
	            #tUDT_Status.InvalidTotalEntriesStored := #iqUDT_FifoHeader.TotalEntriesStored < 0        // The total number of entries is lower than 0
	            OR #iqUDT_FifoHeader.TotalEntriesStored > #iqUDT_FifoHeader.MaxNrOfEntries;               // The total number of entries is greater than the maximum number of entries

	        END_REGION

	        REGION 4.3 – The number of the next entry to write

	            // Set the invalid next entry to write
	            #tUDT_Status.InvalidNextEntryToWrite := #iqUDT_FifoHeader.NextEntryToWrite < 0            // The number of next entry to write is lower than 0
	            OR #iqUDT_FifoHeader.NextEntryToWrite >= #iqUDT_FifoHeader.MaxNrOfEntries;                // The number of next entry to write is greater or equal to the maximum number of entries

	        END_REGION

	        REGION 4.4 – The number of the next entry to read

	            // Set the invalid next entry to read
	            #tUDT_Status.InvalidNextEntryToRead := #iqUDT_FifoHeader.NextEntryToRead < 0              // The number of next entry to read is lower than 0
	            OR #iqUDT_FifoHeader.NextEntryToRead >= #iqUDT_FifoHeader.MaxNrOfEntries;                 // The number of next entry to read is greater or equal to the maximum nr of entries

	        END_REGION

	        REGION 4.5 – FIFO header validation summary

	            // Create collective header error
	            #tx_HeaderValid := NOT #tUDT_Status.InvalidMaxNrOfEntries
	            AND NOT #tUDT_Status.InvalidTotalEntriesStored
	            AND NOT #tUDT_Status.InvalidNextEntryToWrite
	            AND NOT #tUDT_Status.InvalidNextEntryToRead;

	        END_REGION

	    END_IF;

	END_REGION

	REGION 5 – Writing the data into the FIFO buffer

	    IF (#ic_Mode = 'W'                                                                          // Write mode selected
	        AND #tx_HeaderValid                                                                     // FIFO header valid
	        AND NOT #tUDT_Status.InvalidDataType)                                                  // Buffer data type valid
	    THEN


	        IF (#iqUDT_FifoHeader.TotalEntriesStored < #iqUDT_FifoHeader.MaxNrOfEntries)          // Checking total number of stored entries
	        THEN

	            // Move input data to FIFO data buffer
	            #ti_MoveBLKErrorCode := MOVE_BLK_VARIANT(SRC := #iqv_Data,
	                                                     COUNT := 1,
	                                                     SRC_INDEX := 0,
	                                                     DEST_INDEX := #iqUDT_FifoHeader.NextEntryToWrite,
	                                                     DEST => #iqv_DataBuffer);

	            // Increment the number of the next entry to write
	            #iqUDT_FifoHeader.NextEntryToWrite += 1;

	            // Increment the total number of stored entries
	            #iqUDT_FifoHeader.TotalEntriesStored += 1;


	            IF (#iqUDT_FifoHeader.NextEntryToWrite >= #iqUDT_FifoHeader.MaxNrOfEntries)       // Check the number of the next entry to write
	            THEN

	                #iqUDT_FifoHeader.NextEntryToWrite := 0;

	            END_IF;

	        ELSE

	            #tUDT_Status.FifoFull := TRUE;

	        END_IF;

	    END_IF;

	END_REGION

	REGION 6 – Reading the data from the FIFO data buffer

	    IF (#ic_Mode = 'R'                                                                  // Read mode selected
	        AND #tx_HeaderValid                                                             // FIFO header valid
	        AND NOT #tUDT_Status.InvalidDataType)                                           // Buffer data type valid
	    THEN

	        IF (#iqUDT_FifoHeader.TotalEntriesStored > 0)                                   // Checking total number of stored entries
	        THEN

	            // Move the FIFO data to the data output
	            #ti_MoveBLKErrorCode := MOVE_BLK_VARIANT(SRC := #iqv_DataBuffer,
	                                                     COUNT := 1,
	                                                     SRC_INDEX := #iqUDT_FifoHeader.NextEntryToRead,
	                                                     DEST_INDEX := 0,
	                                                     DEST => #iqv_Data);

	            // Increment the number of the next entry to read
	            #iqUDT_FifoHeader.NextEntryToRead += 1;

	            // Decrement the total number of stored entries
	            #iqUDT_FifoHeader.TotalEntriesStored -= 1;

	            IF (#iqUDT_FifoHeader.NextEntryToRead >= #iqUDT_FifoHeader.MaxNrOfEntries)  // Check the number of the next entry to read
	            THEN

	                #iqUDT_FifoHeader.NextEntryToRead := 0;

	            END_IF;

	        END_IF;

	    END_IF;

	END_REGION

	REGION 7 – Clearing the FIFO header

	    IF (#ic_Mode = 'C'                      // Clear mode selected
	        AND #tx_HeaderValid)                // FIFO header valid
	    THEN

	        #iqUDT_FifoHeader.TotalEntriesStored := 0;
	        #iqUDT_FifoHeader.NextEntryToWrite := 0;
	        #iqUDT_FifoHeader.NextEntryToRead := 0;

	    END_IF;

	END_REGION

	REGION 8 – FIFO management status update

	    IF (#tx_HeaderValid)                   // The header is valid
	    THEN

	        REGION 8.1 – FIFO Empty

	            // Set the FIFO empty status bit
	            #iqUDT_FifoHeader.Status.Empty := #iqUDT_FifoHeader.TotalEntriesStored = 0;

	        END_REGION

	        REGION 8.2 – FIFO Full

	            // Set the FIFO full status bit
	            #iqUDT_FifoHeader.Status.Full := #iqUDT_FifoHeader.TotalEntriesStored = #iqUDT_FifoHeader.MaxNrOfEntries;

	        END_REGION

	        REGION 8.3 – FIFO Pre-full

	            IF (#iqUDT_FifoHeader.TotalEntriesStored >= 0.9 * #iqUDT_FifoHeader.MaxNrOfEntries)       // Checking if the number of total stored entries is greater or equal to 90% of the max number of entries
	            THEN

	                // Set the FIFO pre-full status
	                #iqUDT_FifoHeader.Status.Prefull := TRUE;
	                #tUDT_Status.FifoPreFull := TRUE;

	            ELSE

	                #iqUDT_FifoHeader.Status.Prefull := FALSE;

	            END_IF;

	        END_REGION

	    END_IF;

	END_REGION

	REGION 9 – Status

	    REGION 9.1 – Common status update

	        // Collective error output
	        #qx_Error := NOT #tx_HeaderValid
	        OR #tUDT_Status.InvalidMode
	        OR #tUDT_Status.FifoFull
	        OR #tUDT_Status.InvalidDataType;

	        // Collective warning output
	        #qx_Warning := #tUDT_Status.FifoPreFull;

	    END_REGION

	    REGION 9.2 – Status update

	        // Update the outer status structure with internal status structure
	        #qUDT_Status := #tUDT_Status;

	    END_REGION

	END_REGION
END_FUNCTION

DATA_BLOCK "DB_GIN"
TITLE = DB_GIN
{ S7_Optimized_Access := 'TRUE' }
AUTHOR : MHSE
FAMILY : GeneralSystemFunctions
VERSION : 3.0
NON_RETAIN
//Data block to store parcels informations.
   VAR
      GIN { ExternalAccessible := 'False'; ExternalVisible := 'False'; ExternalWritable := 'False'; S7_SetPoint := 'False'} : Array[1..1] of "UDT_GIN";   // GIN informations - for project remove unneeded customers and extend array bound range to 9999
   END_VAR


BEGIN

END_DATA_BLOCK

TYPE "UDT_Message"
TITLE = UDT_Message
VERSION : 0.1
//User-defined structure of the message characters array.
   STRUCT
      Character : Array[0..499] of Char;   // Message character
   END_STRUCT;

END_TYPE

TYPE "UDT_FedExMessageHeader"
VERSION : 0.1
   STRUCT
      STX : Char;
      MessageLength : String[4];
      MessageType : String[2];
   END_STRUCT;

END_TYPE

TYPE "UDT_FedExCustomerID"
VERSION : 0.1
   STRUCT
      CustomerIDMemory { ExternalAccessible := 'False'; ExternalVisible := 'False'; ExternalWritable := 'False'} : DInt;   // Customer ID memory
      CustomerIDReference { ExternalAccessible := 'False'; ExternalVisible := 'False'; ExternalWritable := 'False'} : Array[1..999999] of Int;   // Customer ID reference array
   END_STRUCT;

END_TYPE

TYPE "UDT_Chute3BrakeStatus"
VERSION : 0.1
   STRUCT
      Status { S7_SetPoint := 'True'} : Int;   // Status number
      Specific : Struct   // Chute specific status structure
         ChuteJam : Bool;   // Jam on chute
         ChuteFull : Bool;   // Chute is full
         ChuteHalfFull : Bool;   // Chute is half full
         DisableFromHMI : Bool;   // Disabled from HMI
         DisableFromHLC : Bool;   // Disabled from HLC
         BrakeFaultTop : Bool;   // Top brake bar  is faulty
         BrakeFaultMiddle : Bool;   // Middle brake bar is faulty
         BrakeFaultBottom : Bool;   // Bottom brake bar is faulty
      END_STRUCT;
   END_STRUCT;

END_TYPE

TYPE "UDT_FedExMessagePS"
VERSION : 0.1
   STRUCT
      SystemID : String[15];   // Identifier of the system.
      ParameterID : String[4];   // Parameter code to identify which parameter value is being set
      ParameterValue : String[82];   // New value for the specified parameter
      Timestamp : String[17];   // Local Time Timestamp
      TimeZoneDesignator : String[5];   // Time Zone Designator
   END_STRUCT;

END_TYPE

TYPE "UDT_FedExMessageCD"
VERSION : 0.1
   STRUCT
      CommandCode : String[3];   // Generated during configuration.It is a fixed value for all systems
      CommandValue : String[82];   // System ID of the system making the request.
      Timestamp : String[17];   // Local time timestamp
      TimeZoneDesignator : String[5];   // Time zone designator
   END_STRUCT;

END_TYPE

TYPE "UDT_FedExMessageDaRa"
VERSION : 0.1
   STRUCT
      LLCSystemID : String[15];   // Identifier of Low-Level controls
      PackageID : String[15];   // Number assigned by the LLC system
      HLCPackageID : String[10];   // Unique number for the specific package during it stays in HLC system.
      CellNumber : String[4];   // Tray/Cell number (for loop sorters) or generated by LLC (on line sorters).
      Destination1 : String[6];   // Location code value that describes where the package should go (Diverter Number).
      CutOffTimeDestination1 : String[5];   // Cut Off Time in Local Time.
      Destination2 : String[6];   // Location code value that describes where the package should go (Diverter Number).
      CutOffTimeDestination2 : String[5];   // Cut Off Time in Local Time.
      Destination3 : String[6];   // Location code value that describes where the package should go (Diverter Number).
      CutOffTimeDestination3 : String[5];   // Cut Off Time in Local Time.
      Destination4 : String[6];   // Location code value that describes where the package should go (Diverter Number).
      CutOffTimeDestination4 : String[5];   // Cut Off Time in Local Time.
      Destination5 : String[6];   // Location code value that describes where the package should go (Diverter Number).
      CutOffTimeDestination5 : String[5];   // Cut Off Time in Local Time.
      HLCDataText : String[20];   // Free text for future use.
      Barcodedata : String[50];   // Sortation barcode
      HLCResultCode : String[16];   // Result code based on processing of the scan event messages.
      Timestamp : String[17];   // Local time timestamp
      TimeZoneDesignator : String[5];   // Time zone designator
   END_STRUCT;

END_TYPE

TYPE "UDT_Chute3BrakesConfiguration"
VERSION : 0.1
   STRUCT
      BrakeConfiguration1 { S7_SetPoint := 'False'} : "UDT_PneumaticBrakeConfiguration";   // First brake configuration
      BrakeConfiguration2 { S7_SetPoint := 'False'} : "UDT_PneumaticBrakeConfiguration";   // Secound brake configuration
      StopperConfiguration { S7_SetPoint := 'False'} : "UDT_StopRollerConfiguration";   // Stopper configuration
      PECFullOnDelay : UDInt;   // On delay time PEC full signal
      PECFullOffDelay : UDInt;   // Off delay time PEC full signal
      PECHalfFullOnDelay : UDInt;   // On delay time PEC half full signal
      PECHalfFullOffDelay : UDInt;   // Off delay time PEC half full signal
      PECMiddleOnDelay : UDInt;   // On delay time PEC middle signal
      PECMiddleOffDelay : UDInt;   // Off delay time PEC middle signal
      LongBrakePauseOnDelay : UDInt;   // On delay time from common stop PEC signals
      NumberOfTheEquipment : String[3];   // Number of the equipment 001-999
      "Device ID" : String[6];   // ID of the Device Type
      DEPCOD : String[6];   // Depot Code
      LOConEquipment : String[6];   // Location of the equipment
   END_STRUCT;

END_TYPE

FUNCTION "FC_GetDevicePN" : Void
TITLE = FC_GetDevicePN
{ S7_Optimized_Access := 'TRUE' }
AUTHOR : MHSE
VERSION : 3.0
// ATTRIBUTES
// AUTO_NUMBER = True
// BLOCK_NUMBER = 18
// END_ATTRIBUTES
   VAR_INPUT
      is_PNDeviceName : String;   // Name of the device
      ix_SimulationModeActive : Bool;   // True = Simulation mode active
   END_VAR

   VAR_IN_OUT
      iqUDT_PND : "UDT_PNDevice";   // Device found in Profinet structure
   END_VAR

   VAR_TEMP
      ti_NrOfConfiguredPNNetworks : Int;   // Number of networks configured in project
      ti_NrOfDevices : Int;   // Nr of devices is networks
      ti_LcPNNetworkNumber : Int;   // Loop counter to find PN network number
      ti_LcPNDeviceNumber : Int;   // Loop counter to find PN device number
   END_VAR


BEGIN
	(*
	----------------------------------------------------------------------------------------

	Version history:
	Date        | Version   | Author        | Remark
	----------------------------------------------------------------------------------------
	16/09/2019  | 2.3       | F.Baten       | Cut out of 'FB_RIO'
	29/09/2019  | 2.4       | K.Pokorski    | Network seach started from 1 instead 0
	30/09/2019  | 2.5       | K.Pokorski    | Chagne prefixes of temporary varaibles from 'si' to 'ti'
	12/11/2019  | 3.0       | P.Majka       | 3.0 MHS library release TIA 15.1
	21/02/2023  | 4.0       | F.Baten       | 4.0 Release TIA 17.5
	*)

	REGION 1 - Get Device Profinet number
	    // if simulation is disabled
	    IF NOT #ix_SimulationModeActive
	    THEN
	        // And the profinet device is not found yet
	        IF (#is_PNDeviceName <> "DB_ProfinetDiagnostic".ProfinetNetworks[#iqUDT_PND.PNNetworknumber].DeviceStatus[#iqUDT_PND.PNDeviceNumber].DeviceState.PNDeviceName)
	            OR #iqUDT_PND.PNDeviceFound = FALSE
	        THEN
	            #iqUDT_PND.PNDeviceFound := FALSE;

	            // check how many profinet networks are configured
	            #ti_NrOfConfiguredPNNetworks := "FC_GetNrOfArrayEl"("DB_ProfinetDiagnostic".ProfinetNetworks);

	            FOR #ti_LcPNNetworkNumber := 1 TO (#ti_NrOfConfiguredPNNetworks) DO

	                #iqUDT_PND.PNNetworknumber := #ti_LcPNNetworkNumber;

	                // and check how many devices are configured per network
	                #ti_NrOfDevices := "FC_GetNrOfArrayEl"("DB_ProfinetDiagnostic".ProfinetNetworks[#iqUDT_PND.PNNetworknumber].DeviceStatus);

	                // check for each of the devices in the networks if the PN device name is similair to the configured device name
	                FOR #ti_LcPNDeviceNumber := 0 TO (#ti_NrOfDevices - 1) DO

	                    #iqUDT_PND.PNDeviceNumber := #ti_LcPNDeviceNumber;

	                    // set device found when a match is found for the device name in the PN network
	                    IF (#is_PNDeviceName = "DB_ProfinetDiagnostic".ProfinetNetworks[#iqUDT_PND.PNNetworknumber].DeviceStatus[#iqUDT_PND.PNDeviceNumber].DeviceState.PNDeviceName
	                        AND #is_PNDeviceName <> '')
	                    THEN

	                        #iqUDT_PND.PNDeviceFound := TRUE;
	                        EXIT;

	                    END_IF;
	                END_FOR;

	                // exit loop when device name is matching
	                IF #iqUDT_PND.PNDeviceFound
	                THEN

	                    EXIT;

	                END_IF;
	            END_FOR;
	        END_IF;
	    END_IF;

	END_REGION
END_FUNCTION

FUNCTION "FC_GetPNPortStatus" : Void
{ S7_Optimized_Access := 'TRUE' }
VERSION : 0.1
// ATTRIBUTES
// AUTO_NUMBER = True
// BLOCK_NUMBER = 20
// END_ATTRIBUTES
   VAR_INPUT
      ii_NumberOfPorts : Int;   //  Number of ports in device
      iUDT_DevicePNInfo : "UDT_PNDevice";   //  PN device info structure
   END_VAR

   VAR_OUTPUT
      qa_PortFault : Array[1..8] of Bool;   //  When TRUE then specific port has a fault
   END_VAR

   VAR_TEMP
      tp_GetDiagInfo {InstructionName := 'DIS'; LibVersion := '1.0'} : DIS;   //  Diagnostic structure
      tp_DeviceGeoAddr {InstructionName := 'GEOADDR'; LibVersion := '1.0'} : GEOADDR;   //  Device pointer structre
      ta_PortFault : Array[1..8] of Bool;   //  When TRUE then port has a fault
      ti_Geo2LogStatus : Int;   //  GEO2LOG status code
      ti_GetDiagStatus : Int;   //  Get_Diag status code
      ti_Log2GeoStatus : Int;   //  LOG2GEO status code
      ti_Loopcounter : Int;   //  Loop counter
      tui_cnt : UInt;   //  Not used
      tdi_PortLaddr : HW_ANY;   //  HW identifier
      ti_PortFault : Bool;   //  At least one port is faulty
      tx_ConfigurationError : Bool;   //  Configuration error occurred
   END_VAR

   VAR CONSTANT
      ci_Area : UInt := 1;   //     Area ID of IO Profinet devices
      ci_HWTYPE : UInt := 5;
      ci_PortSlot : UInt := 0;
      ci_PortSubslot : Word := 16#8000;
   END_VAR


BEGIN
	(*
	----------------------------------------------------------------------------------------

	Version history:
	Date        | Version   | Author        | Remark
	----------------------------------------------------------------------------------------
	03/11/2020  | 3.0       | K.Pokorski    | first release MHS TIA 15.1
	17/12/2020  | 3.1       | K.Pokorski    | Run operation only during error
	21/02/2023  | 4.0       | F.Baten       | 4.0 Release TIA 17.5
	*)

	REGION 1 - Check configuration

	    #tx_ConfigurationError := #ii_NumberOfPorts < 1
	    OR #ii_NumberOfPorts > 8
	    OR NOT #iUDT_DevicePNInfo.PNDeviceFound;

	END_REGION

	REGION 2 - Read profinet network number

	    // Using LOG2GEO profinet network address is read
	    #ti_Log2GeoStatus := LOG2GEO(LADDR := "DB_ProfinetDiagnostic".ProfinetNetworks[#iUDT_DevicePNInfo.PNNetworknumber].DeviceStatus[#iUDT_DevicePNInfo.PNDeviceNumber].DeviceState.HW_ID,
	                                 GEOADDR := #tp_DeviceGeoAddr);

	END_REGION

	REGION 3 - Preparation the device pointer

	    // HWTYPE = 5 - Submodule
	    #tp_DeviceGeoAddr.HWTYPE := #ci_HWTYPE;
	    // AREA = 1 - PROFINET IO
	    #tp_DeviceGeoAddr.AREA := #ci_Area;
	    // SLOT = 0 - Ports are on slot 0
	    #tp_DeviceGeoAddr.SLOT := #ci_PortSlot;
	    // STATION - Profinet number
	    #tp_DeviceGeoAddr.STATION := "DB_ProfinetDiagnostic".ProfinetNetworks[#iUDT_DevicePNInfo.PNNetworknumber].DeviceStatus[#iUDT_DevicePNInfo.PNDeviceNumber].DeviceState.ProfinetNumber;

	END_REGION

	REGION 4 - Checking the port status
	    // If device report error and is available on the PN network
	    IF "DB_ProfinetDiagnostic".ProfinetNetworks[#iUDT_DevicePNInfo.PNNetworknumber].DeviceStatus[#iUDT_DevicePNInfo.PNDeviceNumber].DeviceState.Error
	        AND "DB_ProfinetDiagnostic".ProfinetNetworks[#iUDT_DevicePNInfo.PNNetworknumber].DeviceStatus[#iUDT_DevicePNInfo.PNDeviceNumber].DeviceState.Exist
	        AND NOT #tx_ConfigurationError
	    THEN

	        // Loop through all profinet ports
	        FOR #ti_Loopcounter := 1 TO #ii_NumberOfPorts DO
	            // Reset auxiliary port fault bit
	            #ta_PortFault[#ti_Loopcounter] := FALSE;
	            // SUBSLOT = 16#8000 plus port number (TIA structure to refer to port)
	            #tp_DeviceGeoAddr.SUBSLOT := INT_TO_UINT(WORD_TO_INT(#ci_PortSubslot) + (#ti_Loopcounter));
	            // Using GEO2LOG port address is read
	            #ti_Geo2LogStatus := GEO2LOG(GEOADDR := #tp_DeviceGeoAddr, LADDR => #tdi_PortLaddr);
	            // Using GET_DIAG port status is read
	            #ti_GetDiagStatus := GET_DIAG(MODE := 1, LADDR := #tdi_PortLaddr, CNT_DIAG => #tui_cnt, DIAG := #tp_GetDiagInfo);

	            // Set port fault if all operations do not report any error and port is faulty
	            IF #ti_GetDiagStatus = 0
	                AND #ti_Geo2LogStatus = 0
	                AND #ti_Log2GeoStatus = 0
	                AND #tp_GetDiagInfo.OwnState = 4
	            THEN
	                #ta_PortFault[#ti_Loopcounter] := TRUE;
	            END_IF;
	        END_FOR;
	        // Reset module status if error occurred
	    ELSIF #tx_ConfigurationError
	    THEN
	        FOR #ti_Loopcounter := 1 TO 8 DO
	            #ta_PortFault[#ti_Loopcounter] := FALSE;
	        END_FOR;
	    END_IF;

	END_REGION

	REGION 5 - Write output

	    #qa_PortFault := #ta_PortFault;

	END_REGION


END_FUNCTION

TYPE "UDT_Connection"
TITLE = UDT_Connection
VERSION : 0.1
//User-defined structure of connection parameters.
   STRUCT
      ActiveEstablished : Bool := FALSE;   // 0 – Passive connection establishment; 1 – Active connection establishment
      Interface_ID : HW_ANY := 64;   // Interface ID of CPU Ethernet interface
      ID : CONN_OUC;   // Unique ID as system reference for the connection
      IP : Array[1..4] of Int;   // IP address
      Port : UInt;   // Port number of the communication partner
      ConTimeout : DInt;   // Maximum waiting time for response from the communication partner [ms]
   END_STRUCT;

END_TYPE

TYPE "UDT_FedExDestinations"
VERSION : 0.1
   STRUCT
      PhysicalDestination : DInt;
      Destination : Array[0..5] of DInt;   // Destination code to compare to to go to position
   END_STRUCT;

END_TYPE

TYPE "UDT_FedExHeartbeatStatistics"
TITLE = UDT_HeartbeatStatistics
VERSION : 0.1
//User-defined structure of FB_Heartbeat function block statistics.
   STRUCT
      ConLost : UDInt;   // Statistics of connection lost
      MsgNotSent : UDInt;   // Statistics of not send messages when it was requested
   END_STRUCT;

END_TYPE

FUNCTION_BLOCK "FB_FedExCustomerID"
{ S7_Optimized_Access := 'TRUE' }
VERSION : 0.1
// ATTRIBUTES
// AUTO_NUMBER = True
// BLOCK_NUMBER = 64
// END_ATTRIBUTES
   VAR_INPUT
      ii_Gin { ExternalAccessible := 'False'; ExternalVisible := 'False'; ExternalWritable := 'False'} : Int;   // Gin number
   END_VAR

   VAR_IN_OUT
      iqUDT_CustomerID : "UDT_FedExCustomerID";   // Customer ID structure
   END_VAR

   VAR
      si_OldGIN { ExternalAccessible := 'False'; ExternalVisible := 'False'; ExternalWritable := 'False'} : Int;   // Old GIN number
   END_VAR

   VAR_TEMP
      tx_InvalidGIN : Bool;   // Invalid GIN number
   END_VAR


BEGIN
	(*
	----------------------------------------------------------------------------------------

	Version history:
	Date        | Version   | Author        | Remark
	----------------------------------------------------------------------------------------
	30/06/2022  | 0.1       | K.Pokorski    | first release MHS TIA 16
	21/02/2023  | 4.0       | F.Baten       | 4.0 Release TIA 17.5
	*)

	REGION 1 - GIN validation

	    // GIN validation
	    #tx_InvalidGIN :=
	    #ii_Gin < 1
	    OR #ii_Gin > 9999;

	END_REGION

	REGION 2 - Save Customer ID and GIN number

	    IF NOT #tx_InvalidGIN
	    THEN

	        IF #ii_Gin <> #si_OldGIN
	            AND "DB_GIN".GIN[#ii_Gin].FedEx.CustomerID = 0
	        THEN

	            #iqUDT_CustomerID.CustomerIDMemory += 1;
	            IF #iqUDT_CustomerID.CustomerIDMemory > 999999 THEN

	                #iqUDT_CustomerID.CustomerIDMemory := 1;

	            END_IF;


	            #iqUDT_CustomerID.CustomerIDReference[#iqUDT_CustomerID.CustomerIDMemory] := #ii_Gin;
	            "DB_GIN".GIN[#ii_Gin].FedEx.CustomerID := #iqUDT_CustomerID.CustomerIDMemory;


	            #si_OldGIN := #ii_Gin;

	        END_IF;
	    END_IF;
	END_REGION


END_FUNCTION_BLOCK

TYPE "UDT_FedexLoginStatus"
VERSION : 0.1
   STRUCT
      Accepted : Bool;
      Rejected : Bool;
   END_STRUCT;

END_TYPE

TYPE "UDT_ConveyorCommonConfiguration"
VERSION : 0.1
   STRUCT
      Length : DInt;   // Conveyor length [mm]
      LengthCorrection : DInt;   // Length correction [mm]
   END_STRUCT;

END_TYPE

DATA_BLOCK "DB_ExternalGIN"
{ S7_Optimized_Access := 'TRUE' }
VERSION : 0.1
NON_RETAIN
   VAR
      UnexpectedSI { ExternalAccessible := 'False'; ExternalVisible := 'False'; ExternalWritable := 'False'; S7_SetPoint := 'False'} : "UDT_GIN";
   END_VAR


BEGIN

END_DATA_BLOCK

TYPE "UDT_FedExMessageSI"
VERSION : 0.1
   STRUCT
      Header { S7_SetPoint := 'False'} : "UDT_FedExMessageHeader";
      ADCSystemID : String[15];   // Identifier of Automated Data Capture system.
      ScanUnitType : String[1];   // Scan Unit Type
      ImageID : String[6];   // Image ID number (000001 to 999999), token for the parcel created by the ADCsystem.
      PackageID : String[15];   // Number assigned by the LLC system or ADC system
      HLCPackageID : String[10];   // Unique number for the specific package during it stays in HLC system.
      DIMSystemID : String[15];   // Identifier of dimensioning system
      DimStatus : String[5];
      PackageDimLength : String[6];   // Length dimension of package in resolution of dim system.
      PackageDimWidth : String[6];   // Width dimension of package in resolution of dim system.
      PackageDimHeight : String[6];   // Height dimension of package in resolution of dim system.
      DIMUOM : String[2];   // Unit of measure of the package dimensions.
      DimLFTstatusCode : String[8];   // Dimension LFT status code.
      AlibiDims : String[25];   // Alibi for Dimensions
      SCLSystemID : String[15];   // Identifier of weight scale.
      SCLStatus : String[5];   // Basic diagnostic information from the weight scale system.
      SCLWT : String[6];   // Scale weight of package in resolution of scale system.
      SCLWTUOM : String[2];   // Unit of measurement for Weight
      SCLLFTStatusCode : String[2];   // Scale LFT status code.
      AlibiWeight : String[25];   // Alibi for Weight
      Stackable : String[1];   // If stackable recognition is enabled, Y or N
      Timestamp : String[17];   // Local time timestamp
      TimeZoneDesignator : String[5];   // Time zone designator
      Barcode1Identification : String[3];   // Barcode identifier code.
      Barcode1status : String[2];   // Barcode confidence factor
      Barcode1datalength : String[4];   // String length of barcode data in bytes; inclusive of this field. Use 0054 as a fixed value
      Barcode1data : String[50];   // Highest priority barcode
      Barcode2Identification : String[3];   // Barcode identifier code.
      Barcode2status : String[2];   // Barcode confidence factor
      Barcode2datalength : String[4];   // String length of barcode data in bytes; inclusive of this field. Use 0054 as a fixed value
      Barcode2data : String[50];   // Highest priority barcode
      Barcode3Identification : String[3];   // Barcode identifier code.
      Barcode3status : String[2];   // Barcode confidence factor
      Barcode3datalength : String[4];   // String length of barcode data in bytes; inclusive of this field. Use 0054 as a fixed value
      Barcode3data : String[50];   // Highest priority barcode
      TotalBarcodeDataLength : String[4];   // Length of all barcode data that was sent in bytes;
      PackageDataTruncated : String[1];   // Y = Full length of barcode data exceeds 9999 bytes, data truncated
      CameraHeadstatus : String[2];   // Diagnostic information on camera/laser heads performing barcode reads.
   END_STRUCT;

END_TYPE

TYPE "UDT_FedExMessageLoginResponse"
VERSION : 0.1
   STRUCT
      Header { S7_SetPoint := 'False'} : "UDT_FedExMessageHeader";
      FacilityID : String[8];   // Generated during configuration.It is a fixed value for all systems
      SystemID : String[15];   // System ID of the system making the request.
      VersionID : String[6];   // Interface document version.
      ConnectionStatus : String[1];   // Y=Succes, N=Failure
      LocalHost : String[32];   // IP Address of the existing connection. If this is the first connection, IP Address or Hostname of the connecting host.
   END_STRUCT;

END_TYPE

TYPE "UDT_FedExMessageWS"
VERSION : 0.1
   STRUCT
      Header { S7_SetPoint := 'False'} : "UDT_FedExMessageHeader";
      SCLSystemID : String[15];   // Identifier of weight scale.
      PackageID : String[15];   // Number assigned by the LLC system
      SCLWT : String[6];   // Scale weight of package in resolution of scale system.
      SCLWTUOM : String[2];   // Unit of measurement for Weight
      SCLLFTStatusCode : String[2];   // Scale LFT status code.
      AlibiWeight : String[25];   // Alibi for Weight
      Timestamp : String[17];   // Local time timestamp
      TimeZoneDesignator : String[5];   // Time zone designator
   END_STRUCT;

END_TYPE

TYPE "UDT_TCPIPReceiveStatistics"
TITLE = UDT_TCPIPReceiveStatistics
VERSION : 0.1
//User-defined structure of FB_TCPIPReceive function block statistics.
   STRUCT
      InvalidMsg : UInt;   // Invalid message received
   END_STRUCT;

END_TYPE

TYPE "UDT_VfdKebaSystemStatistics"
VERSION : 0.1
   STRUCT
      PNSlaveNotOnline : "UDT_EventStatistic";   // Statistics of Profinet slave not online
      PNSlaveError : "UDT_EventStatistic";   // Statistics of a Profinet slave error
      Ax1InternalError : "UDT_EventStatistic";   // Statistics of an axis 1 internal error
      Ax2InternalError : "UDT_EventStatistic";   // Statistics of an axis 2 internal error
      CommunicationError : "UDT_EventStatistic";   // Statistics of a communication error
      Ax1Running : "UDT_EventStatistic";   // Statistics for axis 1 running time
      Ax2Running : "UDT_EventStatistic";   // Statistics for axis 2 running time
   END_STRUCT;

END_TYPE

TYPE "UDT_FedExCommands"
VERSION : 0.1
   STRUCT
      StartSort : Struct   // Sent to LLC to designate the Sort has started. – Functionality to include reset of LLC Application buffers from previous sort
         NewMessage : Bool;   // New message received from UDS
         StartSort : Bool;   // Sent to LLC to designate the Sort has started. – Functionality to include reset of LLC Application buffers from previous sort
      END_STRUCT;
      EndSort : Struct   // Sent to LLC to designate the Sort has stopped. This message should not clear LLC counters. To be used in future cases.
         NewMessage : Bool;   // New message received from UDS
         EndSort : Bool;   // Sent to LLC to designate the Sort has stopped. This message should not clear LLC counters. To be used in future cases.
      END_STRUCT;
      UploadChuteStatus : Struct   // Sent to LLC so HLC can receive an update of all the current chute status. This information is required to work in optimal conditions when chute grouping has been enabled.
         NewMessage : Bool;   // New message received from UDS
      END_STRUCT;
      UploadAllStatus : Struct   // Sent to LLC so HLC can receive an update of the current equipment status.
         NewMessage : Bool;   // New message received from UDS
      END_STRUCT;
      BlockDivertSmalls : Struct   // Divert Block sent to the LLC when a bag is determined Full by the HLC, when a bag must be closed at the beginning of a sort, and to prevent miss-sorts during assignment changes. (Automated Smalls Only)
         NewMessage : Bool;   // New message received from UDS
         SorterNumber : String[5];   // Sorter number
         DivertNumber : String[6];   // Diverter number
      END_STRUCT;
      UnblockDivertSmalls : Struct   // Divert Unblock sent to the LLC when a bag is determined Full by the HLC, when a bag must be closed at the beginning of a sort, and to prevent miss-sorts during assignment changes. (Automated Smalls Only)
         NewMessage : Bool;   // New message received from UDS
         SorterNumber : String[5];   // Sorter number
         DivertNumber : String[6];   // Diverter number
      END_STRUCT;
      EnablePurge : Struct   // Purge Enable command including up to five chutes sent to the LLC when an Operator enables Purge on the HLC.
         NewMessage : Bool;   // New message received from UDS
         PLC : String[6];   // PLC Number
         Chute : Array[1..5] of String;   // Chute number
      END_STRUCT;
      DisablePurge : Struct   // Purge disable command including up to five chutes sent to the LLC when an Operator enables Purge on the HLC.
         NewMessage : Bool;   // New message received from UDS
         PLC : String[6];   // PLC Number
         Chute : Array[1..5] of String[6];   // Chute number
      END_STRUCT;
      ChuteLamp : Struct   // Lamp on the chutes control from HLC
         NewMessage : Bool;   // New message received from UDS
         ChuteNumber : String[6];   // Chute number to control lamp.
         Mode : String[1];   // 0=Off, 1=On, 2=Slow blink, 3=Blink, 4=Fast blink
         Color : String[9];   // 1= Red, 2=Green, 3=Orange
      END_STRUCT;
   END_STRUCT;

END_TYPE

TYPE "UDT_PolisorterInterface"
TITLE = UDT_VSUInterface
VERSION : 0.1
//User-defined structure of VSU interface parameters.
   STRUCT
      Decisionpoint : Int;   // Point in tracking where the destination is found on the Polisorter conveyor [cm]
      RequestedPosition : Int;   // Position requested by destination block
      PositionSetpoint : Int;   // Position number (as configured) to go to by positioning device
      PositionActual : Int;   // Position number the positioning device is actually on
      SwitchingTime : UInt;   // Time it takes to go from one position to the next [ms]
      PNDeviceOk : Bool;   // Device ok
      Automatic : Bool;   // Automatic mode request
      RunEnabled : Bool;   // Running of the positioning device is enabled
      GoReference : Bool;   // Activate reference run
      Referenced : Bool;   // Positioning device is referenced
      Manual : Bool;   // Manual mode request
      Reference_command : Bool;   // Refference command
      JogLeft : Bool;   // Jog request to move equipment left
      JogRight : Bool;   // Jog request to move equipment right
      Ready : Bool;   // Positioning block is running and error free
      MotorRunning : Bool;   // Motor is running
      Positioning : Bool;   // Positioning device is moving to its position
      ResetStatistics : Bool;   // Reset statistics
      InternalErrorVFD : Bool;   // Positioning device internal error
      InternalWarningVFD : Bool;   // Positioning device has a warning
      InternalErrorReset : Bool;   // Reset internal faults
      RequestDieBackUpstream : Bool;   // External request die back to the upstream conveyor of the Polisorter
      ExternalHold : Bool;   // External request to stop the conveyor
      MaintenanceMode : Bool;   // Maitenance mode enabled
      BypassMode : Bool;   // Bypass mode enable
   END_STRUCT;

END_TYPE

TYPE "UDT_XBSChuteInterfaceSend"
VERSION : 0.1
   STRUCT
      ReadyToReceive : Bool;   // Chute is ready to receive
      Running : Bool;   // Downstream line is running
      Fault : Bool;   // Fault on the downstream line
      Warning : Bool;   // Warning on the downstream line
      HalfFull : Bool;   // Chute is half full
      Full : Bool;   // Chute is Full
   END_STRUCT;

END_TYPE

TYPE "UDT_Chute3BrakeStatistics"
VERSION : 0.1
   STRUCT
      ChuteFull : "UDT_EventStatistic";   // Chute full statistics
      ChuteJam : "UDT_EventStatistic";   // Chute jam statistics
      ChuteHalfFull : "UDT_EventStatistic";   // Chute half full statistics
      DisableFromHMI : "UDT_EventStatistic";   // Disable from HMI statistics
      DisableFromHLC : "UDT_EventStatistic";   // Disable from HLC statistics
   END_STRUCT;

END_TYPE

TYPE "UDT_ConveyorHandshake"
TITLE = UDT_ConveyorHandshake
VERSION : 0.1
//User-defined structure of conveyor handshake variables.
   STRUCT
      GIN : Int;   // General identification number
      NrOfPosToShift : Int;   // Number of positions to shift
      DownstreamDisplacement : Int;   // Displacement from downstream [cm]
      RTS { ExternalAccessible := 'False'; ExternalVisible := 'False'; ExternalWritable := 'False'} : Bool;   // Conveyor ready to send
      RTR { ExternalAccessible := 'False'; ExternalVisible := 'False'; ExternalWritable := 'False'} : Bool;   // Conveyor ready to receive
      TIP { ExternalAccessible := 'False'; ExternalVisible := 'False'; ExternalWritable := 'False'} : Bool;   // Transfer in progress
      ResetEnergySave { ExternalAccessible := 'False'; ExternalVisible := 'False'; ExternalWritable := 'False'} : Bool;   // Reset energy save mode
      CascadeStartUp { ExternalAccessible := 'False'; ExternalVisible := 'False'; ExternalWritable := 'False'} : Bool;   // Cascade startup
      ReqStop { ExternalAccessible := 'False'; ExternalVisible := 'False'; ExternalWritable := 'False'} : Bool;   // Request stop
   END_STRUCT;

END_TYPE

TYPE "UDT_Chute3BrakeCommand"
VERSION : 0.1
   STRUCT
      DisableFromHMI : Bool;   // Disable from HMI
      DisableFromHLC : Bool;   // Disable from HLC
   END_STRUCT;

END_TYPE

FUNCTION "FC_FedExDecodeHeader" : Void
{ S7_Optimized_Access := 'TRUE' }
VERSION : 0.1
// ATTRIBUTES
// AUTO_NUMBER = True
// BLOCK_NUMBER = 36
// END_ATTRIBUTES
   VAR_INPUT
      iUDT_FifoMsg : "UDT_Message";   // Buffer for FIFO's message
   END_VAR

   VAR_OUTPUT
      qUDT_MSGHeader : "UDT_FedExMessageHeader";   // Messade header structure
   END_VAR


BEGIN
	(*
	----------------------------------------------------------------------------------------

	Version history:
	Date        | Version   | Author        | Remark
	----------------------------------------------------------------------------------------
	27/10/2021  | 0.1       | J.Krawczuk    | first release MHS TIA 15.1
	18/11/2021  | 0.2       | M.Piela       | Interface changes
	*)

	REGION - 1 Header decode

	    #qUDT_MSGHeader.STX := #iUDT_FifoMsg.Character[0];

	    Chars_TO_Strg(Chars := #iUDT_FifoMsg.Character,
	                  pChars := 1,
	                  Cnt := 0,
	                  Strg => #qUDT_MSGHeader.MessageLength);

	    Chars_TO_Strg(Chars := #iUDT_FifoMsg.Character,
	                  pChars := 5,
	                  Cnt := 0,
	                  Strg => #qUDT_MSGHeader.MessageType);

	END_REGION



END_FUNCTION

TYPE "UDT_ConveyorInterface"
TITLE = UDT_ConveyorInterface
VERSION : 0.1
//User-defined structure of conveyor interface variables.
   STRUCT
      Displacement : Int;   // Displacement per PLC scan [cm] either from position (if available) or speed and time
      SpeedSetpoint : Int;   // Conveyor speed setpoint [mm/s]
      ActualSpeed : Int;   // Conveyors actual speed [mm/s]
      DeltaPosition : Int;   // Read from Conveyor Servo Position [mm] after 1 PLC cycle
      RunFwd { ExternalAccessible := 'False'; ExternalVisible := 'False'; ExternalWritable := 'False'} : Bool;   // Run forward request
      RunRvs { ExternalAccessible := 'False'; ExternalVisible := 'False'; ExternalWritable := 'False'} : Bool;   // Run reverse request
      InternalErrorEncoder { ExternalAccessible := 'False'; ExternalVisible := 'False'; ExternalWritable := 'False'} : Bool;   // Encoder has an error
      InternalErrorVFD { ExternalAccessible := 'False'; ExternalVisible := 'False'; ExternalWritable := 'False'} : Bool;   // VFD has an error
      InternalErrorTracking { ExternalAccessible := 'False'; ExternalVisible := 'False'; ExternalWritable := 'False'} : Bool;   // Tracking has an error
      InternalErrorPEC { ExternalAccessible := 'False'; ExternalVisible := 'False'; ExternalWritable := 'False'} : Bool;   // PEC has an error
      InternalWarningVFD { ExternalAccessible := 'False'; ExternalVisible := 'False'; ExternalWritable := 'False'} : Bool;   // VFD has a warning
      InternalWarningTracking { ExternalAccessible := 'False'; ExternalVisible := 'False'; ExternalWritable := 'False'} : Bool;   // Tracking has a warning
      InternalErrorReset { ExternalAccessible := 'False'; ExternalVisible := 'False'; ExternalWritable := 'False'} : Bool;   // Reset internal errors
      ConfigurationError { ExternalAccessible := 'False'; ExternalVisible := 'False'; ExternalWritable := 'False'} : Bool;   // Configuration error is active
      VFDRunning { ExternalAccessible := 'False'; ExternalVisible := 'False'; ExternalWritable := 'False'} : Bool;   // Motor is running
      VFDatSpeed { ExternalAccessible := 'False'; ExternalVisible := 'False'; ExternalWritable := 'False'} : Bool;   // Motor at speed setpoint
      Disconnected { ExternalAccessible := 'False'; ExternalVisible := 'False'; ExternalWritable := 'False'} : Bool;   // VFD disconnected
      ManualModeActive { ExternalAccessible := 'False'; ExternalVisible := 'False'; ExternalWritable := 'False'} : Bool;   // Covneyor is in manual mode
      ResetStatistics { ExternalAccessible := 'False'; ExternalVisible := 'False'; ExternalWritable := 'False'} : Bool;   // Reset statistics
      HardwareOk { ExternalAccessible := 'False'; ExternalVisible := 'False'; ExternalWritable := 'False'} : Bool;   // Hardware for the Equipment is available and healthy
   END_STRUCT;

END_TYPE

FUNCTION_BLOCK "FB_StopRoller"
{ S7_Optimized_Access := 'TRUE' }
VERSION : 0.1
// ATTRIBUTES
// AUTO_NUMBER = True
// BLOCK_NUMBER = 229
// END_ATTRIBUTES
   VAR_INPUT
      iUDT_StopRollerConfiguration { ExternalAccessible := 'False'; ExternalVisible := 'False'; ExternalWritable := 'False'} : "UDT_StopRollerConfiguration";   // Stop roller configuration structure
      ix_Pressure { ExternalAccessible := 'False'; ExternalVisible := 'False'; ExternalWritable := 'False'} : Bool;   // TRUE when pressure buildup starts
      ix_PECBrake { ExternalAccessible := 'False'; ExternalVisible := 'False'; ExternalWritable := 'False'} : Bool;   // TRUE when the brake photoye is not blocked
      ix_PECStop { ExternalAccessible := 'False'; ExternalVisible := 'False'; ExternalWritable := 'False'} : Bool;   // TRUE when the stop photoye is not blocked
      ix_DownstreamStopActive { ExternalAccessible := 'False'; ExternalVisible := 'False'; ExternalWritable := 'False'} : Bool;   // TRUE when the downstream stop is active
      ix_SafetyOk { ExternalAccessible := 'False'; ExternalVisible := 'False'; ExternalWritable := 'False'} : Bool;   // TRUE when safety is ok
      ix_BrakePauseLong { ExternalAccessible := 'False'; ExternalVisible := 'False'; ExternalWritable := 'False'} : Bool;   // TRUE when receiving a delayed signal to increase brake pause
   END_VAR

   VAR_OUTPUT
      qx_Valve { ExternalAccessible := 'False'; ExternalVisible := 'False'; ExternalWritable := 'False'} : Bool;   // TRUE when valve is activated
      qx_StopActive { ExternalAccessible := 'False'; ExternalVisible := 'False'; ExternalWritable := 'False'} : Bool;   // TRUE when stop is activated to upstream
   END_VAR

   VAR_IN_OUT
      iqUDT_EquipmentControl : "UDT_EquipmentControl";   // Equipment control structure
   END_VAR

   VAR
      s_PECBreakTimerOnOffDelay { ExternalAccessible := 'False'; ExternalVisible := 'False'; ExternalWritable := 'False'; S7_SetPoint := 'False'} : "FB_TimerOnOffDelay";   // Function block to generate on/off signal delay on the brake PEC
      s_PECStopTimerOnOffDelay { ExternalAccessible := 'False'; ExternalVisible := 'False'; ExternalWritable := 'False'; S7_SetPoint := 'False'} : "FB_TimerOnOffDelay";   // Function block to generate on/off signal delay on the Stop PEC
      s_PECPressureTimerOnOffDelay { ExternalAccessible := 'False'; ExternalVisible := 'False'; ExternalWritable := 'False'; S7_SetPoint := 'False'} : "FB_TimerOnOffDelay";   // Function block to generate on/off signal delay on the pressure PEC
      s_StopFunctionTimerOnOffDelay { ExternalAccessible := 'False'; ExternalVisible := 'False'; ExternalWritable := 'False'; S7_SetPoint := 'False'} : "FB_TimerOnOffDelay";   // Function block to generate on/off signal delay on the downstream stop active
      slr_StepTimer { ExternalAccessible := 'False'; ExternalVisible := 'False'; ExternalWritable := 'False'} : LReal;   // Step timer
      si_BrakeFunction { ExternalAccessible := 'False'; ExternalVisible := 'False'; ExternalWritable := 'False'} : Int;   // Brake function step
      sx_PECBrakeFiltered { ExternalAccessible := 'False'; ExternalVisible := 'False'; ExternalWritable := 'False'} : Bool;   // PEC filtered signal
      sx_PECStopFiltered { ExternalAccessible := 'False'; ExternalVisible := 'False'; ExternalWritable := 'False'} : Bool;   // PEC filtered signal
      sx_PECPressureFiltered { ExternalAccessible := 'False'; ExternalVisible := 'False'; ExternalWritable := 'False'} : Bool;   // PEC filtered signal
      sx_DownstreamStop { ExternalAccessible := 'False'; ExternalVisible := 'False'; ExternalWritable := 'False'} : Bool;   // Downstream is stopped
      sx_StopFunctionActive { ExternalAccessible := 'False'; ExternalVisible := 'False'; ExternalWritable := 'False'} : Bool;   // Stop function is activated
      sx_StopRoller { ExternalAccessible := 'False'; ExternalVisible := 'False'; ExternalWritable := 'False'} : Bool;   // Roller is stop
   END_VAR


BEGIN
	(*
	----------------------------------------------------------------------------------------

	Version history:
	Date        | Version   | Author        | Remark
	----------------------------------------------------------------------------------------
	23/06/2021  | 0.0       | F. Baten      | first release TIA 15.1
	20/10/2021  | 0.1       | M. Piela      | Activate valve when system is stoped. Stylistic correction
	21/02/2023  | 4.0       | F.Baten       | 4.0 Release TIA 17.5
	 *)

	REGION 1 - Timers

	    // Filtering brake photo eye signal
	    #s_PECBreakTimerOnOffDelay(iudi_OnDelayTime := #iUDT_StopRollerConfiguration.PECBrakeOnDelay,
	                               iudi_OffDelayTime := #iUDT_StopRollerConfiguration.PECBrakeOffDelay,
	                               ix_SignalToDelay := #ix_PECBrake,
	                               ix_Enable := TRUE,
	                               qx_DelayedSignal => #sx_PECBrakeFiltered);

	    // Filtering stop photo eye signal
	    #s_PECStopTimerOnOffDelay(iudi_OnDelayTime := #iUDT_StopRollerConfiguration.PECStopOnDelay,
	                              iudi_OffDelayTime := #iUDT_StopRollerConfiguration.PECStopOffDelay,
	                              ix_SignalToDelay := #ix_PECStop,
	                              ix_Enable := TRUE,
	                              qx_DelayedSignal => #sx_PECStopFiltered);

	    // Filtering downstream stop photo eye signal
	    #s_StopFunctionTimerOnOffDelay(iudi_OnDelayTime := #iUDT_StopRollerConfiguration.StopFunctionOnDelay,
	                                   iudi_OffDelayTime := #iUDT_StopRollerConfiguration.StopFunctionOffDelay,
	                                   ix_SignalToDelay := #ix_DownstreamStopActive,
	                                   ix_Enable := TRUE,
	                                   qx_DelayedSignal => #sx_DownstreamStop);
	    // Sequence Timer
	    IF #slr_StepTimer > 0
	    THEN
	        #slr_StepTimer -= "DB_Memory".PrevCycleTime;
	        IF #slr_StepTimer < 0
	        THEN
	            #slr_StepTimer := 0;
	        END_IF;
	    END_IF;

	END_REGION

	REGION 2 - Stop roller

	    // Stop roller comes up when outfeed is not active and will fill up until last PEC is occupied.
	    // Sequence
	    // UP
	    IF (#si_BrakeFunction = 0) AND (#slr_StepTimer = 0)
	    THEN
	        #sx_StopRoller := True;
	        #slr_StepTimer := #iUDT_StopRollerConfiguration.BrakePuls;
	        #si_BrakeFunction := 1;
	    END_IF;

	    // Down
	    IF (#si_BrakeFunction = 1) AND (#slr_StepTimer = 0) AND #ix_SafetyOk
	        AND ((#ix_DownstreamStopActive AND #sx_PECStopFiltered AND NOT #sx_PECBrakeFiltered)
	        OR (NOT #ix_DownstreamStopActive AND NOT #sx_PECBrakeFiltered))

	    THEN
	        #sx_StopRoller := False;

	        IF #ix_BrakePauseLong
	        THEN
	            #slr_StepTimer := #iUDT_StopRollerConfiguration.BrakePauseLong;
	        ELSE
	            #slr_StepTimer := #iUDT_StopRollerConfiguration.BrakePause;
	        END_IF;

	        #si_BrakeFunction := 0;
	    END_IF;

	END_REGION

	REGION 3 - Stop roller valve

	    IF #sx_StopFunctionActive AND #sx_PECStopFiltered
	    THEN
	        #sx_StopFunctionActive := FALSE;
	    END_IF;

	    IF #ix_DownstreamStopActive //#sx_PECBrakeFiltered
	    THEN
	        #sx_StopFunctionActive := TRUE;
	    END_IF;

	    IF #iUDT_StopRollerConfiguration.FailSafe
	    THEN
	        #qx_Valve := NOT (#sx_StopRoller OR NOT #ix_SafetyOk) OR #iqUDT_EquipmentControl.Command.Stop;
	    ELSE
	        #qx_Valve := #sx_StopRoller AND #ix_SafetyOk OR #iqUDT_EquipmentControl.Command.Stop;
	    END_IF;

	END_REGION

	REGION 4 - Stop active

	    #qx_StopActive := #sx_StopFunctionActive AND NOT #sx_PECStopFiltered AND NOT #sx_PECBrakeFiltered;

	END_REGION
END_FUNCTION_BLOCK

